LIN {X 0,Y 460.751,Z 770.991,A -85,B 0,C 180,E1 -8393.678,E2 -8393.678} C_VEL
LIN {X 0,Y 461.755,Z 759.273,A -85,B 0,C 180,E1 -8394.503,E2 -8394.503} C_VEL
LIN {X 0,Y 462.708,Z 747.249,A -85,B 0,C 180,E1 -8395.228,E2 -8395.228} C_VEL
LIN {X 0,Y 463.653,Z 734.036,A -85,B 0,C 180,E1 -8395.895,E2 -8395.895} C_VEL
LIN {X 0,Y 464.466,Z 720.83,A -85,B 0,C 180,E1 -8396.438,E2 -8396.438} C_VEL
LIN {X 0,Y 465.142,Z 708.707,A -85,B 0,C 180,E1 -8396.832,E2 -8396.832} C_VEL
LIN {X 0,Y 465.664,Z 695.09,A -85,B 0,C 180,E1 -8397.167,E2 -8397.167} C_VEL
LIN {X 0,Y 466.448,Z 652.564,A -85,B 0,C 180,E1 -8397.875,E2 -8397.875} C_VEL
LIN {X 0,Y 468.618,Z 514.421,A -85,B 0,C 180,E1 -8400.1,E2 -8400.1} C_VEL
LIN {X 0,Y 460.454,Z 482.125,A -85,B 0,C 180,E1 -8401.269,E2 -8401.269} C_VEL
LIN {X 0,Y 460.493,Z 480.391,A -85,B 0,C 180,E1 -8401.488,E2 -8401.488} C_VEL
LIN {X 0,Y 460.182,Z 477.208,A -85,B 0,C 180,E1 -8402.052,E2 -8402.052} C_VEL
LIN {X 0,Y 456.778,Z 463.456,A -85,B 0,C 180,E1 -8404.699,E2 -8404.699} C_VEL
LIN {X 0,Y 453.504,Z 451.445,A -85,B 0,C 180,E1 -8407.184,E2 -8407.184} C_VEL
LIN {X 0,Y 453.456,Z 451.209,A -85,B 0,C 180,E1 -8408.311,E2 -8408.311} C_VEL
LIN {X 0,Y 453.489,Z 451.249,A -85,B 0,C 180,E1 -8410.608,E2 -8410.608} C_VEL
LIN {X 0,Y 453.45,Z 451.247,A -85,B 0,C 180,E1 -8413.243,E2 -8413.243} C_VEL
LIN {X 0,Y 453.471,Z 451.237,A -85,B 0,C 180,E1 -8415.78,E2 -8415.78} C_VEL
LIN {X 0,Y 453.486,Z 451.245,A -85,B 0,C 180,E1 -8418.21,E2 -8418.21} C_VEL
LIN {X 0,Y 453.524,Z 451.233,A -85,B 0,C 180,E1 -8420.787,E2 -8420.787} C_VEL
LIN {X 0,Y 453.45,Z 451.238,A -85,B 0,C 180,E1 -8423.917,E2 -8423.917} C_VEL
LIN {X 0,Y 453.476,Z 451.243,A -85,B 0,C 180,E1 -8427.151,E2 -8427.151} C_VEL
LIN {X 0,Y 453.507,Z 451.223,A -85,B 0,C 180,E1 -8430.271,E2 -8430.271} C_VEL
LIN {X 0,Y 453.506,Z 451.227,A -85,B 0,C 180,E1 -8433.294,E2 -8433.294} C_VEL
LIN {X 0,Y 453.496,Z 451.244,A -85,B 0,C 180,E1 -8436.238,E2 -8436.238} C_VEL
LIN {X 0,Y 453.473,Z 451.215,A -85,B 0,C 180,E1 -8439.117,E2 -8439.117} C_VEL
LIN {X 0,Y 453.502,Z 451.225,A -85,B 0,C 180,E1 -8441.944,E2 -8441.944} C_VEL
LIN {X 0,Y 453.531,Z 451.237,A -85,B 0,C 180,E1 -8444.726,E2 -8444.726} C_VEL
LIN {X 0,Y 453.552,Z 451.239,A -85,B 0,C 180,E1 -8448.379,E2 -8448.379} C_VEL
LIN {X 0,Y 453.643,Z 451.216,A -85,B 0,C 180,E1 -8451.985,E2 -8451.985} C_VEL
LIN {X 0,Y 453.663,Z 451.222,A -85,B 0,C 180,E1 -8454.667,E2 -8454.667} C_VEL
LIN {X 0,Y 453.757,Z 451.205,A -85,B 0,C 180,E1 -8457.337,E2 -8457.337} C_VEL
LIN {X 0,Y 453.814,Z 451.204,A -85,B 0,C 180,E1 -8460,E2 -8460} C_VEL
LIN {X 0,Y 453.757,Z 451.208,A -85,B 0,C 180,E1 -8462.663,E2 -8462.663} C_VEL
LIN {X 0,Y 453.671,Z 451.213,A -85,B 0,C 180,E1 -8466.225,E2 -8466.225} C_VEL
LIN {X 0,Y 453.584,Z 451.232,A -85,B 0,C 180,E1 -8468.913,E2 -8468.913} C_VEL
LIN {X 0,Y 453.554,Z 451.233,A -85,B 0,C 180,E1 -8472.529,E2 -8472.529} C_VEL
LIN {X 0,Y 453.535,Z 451.228,A -85,B 0,C 180,E1 -8476.196,E2 -8476.196} C_VEL
LIN {X 0,Y 453.511,Z 451.24,A -85,B 0,C 180,E1 -8479.041,E2 -8479.041} C_VEL
LIN {X 0,Y 453.467,Z 451.245,A -85,B 0,C 180,E1 -8481.836,E2 -8481.836} C_VEL
LIN {X 0,Y 453.505,Z 451.229,A -85,B 0,C 180,E1 -8484.735,E2 -8484.735} C_VEL
LIN {X 0,Y 453.53,Z 451.223,A -85,B 0,C 180,E1 -8487.961,E2 -8487.961} C_VEL
LIN {X 0,Y 453.475,Z 451.25,A -85,B 0,C 180,E1 -8490.759,E2 -8490.759} C_VEL
LIN {X 0,Y 453.469,Z 451.216,A -85,B 0,C 180,E1 -8493.913,E2 -8493.913} C_VEL
LIN {X 0,Y 453.464,Z 451.253,A -85,B 0,C 180,E1 -8497.188,E2 -8497.188} C_VEL
LIN {X 0,Y 453.525,Z 451.244,A -85,B 0,C 180,E1 -8499.445,E2 -8499.445} C_VEL
LIN {X 0,Y 453.485,Z 451.249,A -85,B 0,C 180,E1 -8502.992,E2 -8502.992} C_VEL
LIN {X 0,Y 453.458,Z 451.251,A -85,B 0,C 180,E1 -8505.779,E2 -8505.779} C_VEL
LIN {X 0,Y 453.509,Z 451.247,A -85,B 0,C 180,E1 -8509.406,E2 -8509.406} C_VEL
LIN {X 0,Y 453.47,Z 451.248,A -85,B 0,C 180,E1 -8512.223,E2 -8512.223} C_VEL
LIN {X 0,Y 453.483,Z 451.25,A -85,B 0,C 180,E1 -8515.223,E2 -8515.223} C_VEL
LIN {X 0,Y 453.461,Z 451.248,A -85,B 0,C 180,E1 -8518.475,E2 -8518.475} C_VEL
LIN {X 0,Y 453.532,Z 451.242,A -85,B 0,C 180,E1 -8522.039,E2 -8522.039} C_VEL
LIN {X 0,Y 453.51,Z 451.246,A -85,B 0,C 180,E1 -8525.266,E2 -8525.266} C_VEL
LIN {X 0,Y 453.476,Z 451.246,A -85,B 0,C 180,E1 -8528.415,E2 -8528.415} C_VEL
LIN {X 0,Y 453.518,Z 451.244,A -85,B 0,C 180,E1 -8531.009,E2 -8531.009} C_VEL
LIN {X 0,Y 453.564,Z 451.238,A -85,B 0,C 180,E1 -8533.88,E2 -8533.88} C_VEL
LIN {X 0,Y 453.598,Z 451.234,A -85,B 0,C 180,E1 -8537.472,E2 -8537.472} C_VEL
LIN {X 0,Y 453.589,Z 451.233,A -85,B 0,C 180,E1 -8541.087,E2 -8541.087} C_VEL
LIN {X 0,Y 453.633,Z 451.228,A -85,B 0,C 180,E1 -8543.099,E2 -8543.099} C_VEL
LIN {X 0,Y 452.948,Z 451.315,A -85,B 0,C 180,E1 -8543.839,E2 -8543.839} C_VEL
LIN {X 0,Y 450.001,Z 451.681,A -85,B 0,C 180,E1 -8545.041,E2 -8545.041} C_VEL
LIN {X 0,Y 447.578,Z 451.985,A -85,B 0,C 180,E1 -8546.01,E2 -8546.01} C_VEL
LIN {X 0,Y 446.642,Z 452.099,A -85,B 0,C 180,E1 -8546.761,E2 -8546.761} C_VEL
LIN {X 0,Y 446.623,Z 452.101,A -85,B 0,C 180,E1 -8547.014,E2 -8547.014} C_VEL
LIN {X 0,Y 446.791,Z 452.084,A -85,B 0,C 180,E1 -8550,E2 -8550} C_VEL
LIN {X 0,Y 446.706,Z 452.093,A -85,B 0,C 180,E1 -8552.705,E2 -8552.705} C_VEL
LIN {X 0,Y 446.643,Z 452.1,A -85,B 0,C 180,E1 -8556.324,E2 -8556.324} C_VEL
LIN {X 0,Y 446.535,Z 452.112,A -85,B 0,C 180,E1 -8559.055,E2 -8559.055} C_VEL
LIN {X 0,Y 446.53,Z 452.113,A -85,B 0,C 180,E1 -8562.729,E2 -8562.729} C_VEL
LIN {X 0,Y 446.486,Z 452.122,A -85,B 0,C 180,E1 -8566.459,E2 -8566.459} C_VEL
LIN {X 0,Y 446.465,Z 452.122,A -85,B 0,C 180,E1 -8569.303,E2 -8569.303} C_VEL
LIN {X 0,Y 446.414,Z 452.131,A -85,B 0,C 180,E1 -8572.199,E2 -8572.199} C_VEL
LIN {X 0,Y 446.453,Z 452.122,A -85,B 0,C 180,E1 -8575.152,E2 -8575.152} C_VEL
LIN {X 0,Y 446.479,Z 452.122,A -85,B 0,C 180,E1 -8578.178,E2 -8578.178} C_VEL
LIN {X 0,Y 446.414,Z 452.127,A -85,B 0,C 180,E1 -8581.775,E2 -8581.775} C_VEL
LIN {X 0,Y 446.425,Z 452.128,A -85,B 0,C 180,E1 -8584.522,E2 -8584.522} C_VEL
LIN {X 0,Y 446.43,Z 452.127,A -85,B 0,C 180,E1 -8588.082,E2 -8588.082} C_VEL
LIN {X 0,Y 446.436,Z 452.126,A -85,B 0,C 180,E1 -8590.92,E2 -8590.92} C_VEL
LIN {X 0,Y 446.394,Z 452.129,A -85,B 0,C 180,E1 -8593.846,E2 -8593.846} C_VEL
LIN {X 0,Y 446.439,Z 452.126,A -85,B 0,C 180,E1 -8596.397,E2 -8596.397} C_VEL
LIN {X 0,Y 446.461,Z 452.12,A -85,B 0,C 180,E1 -8599.805,E2 -8599.805} C_VEL
LIN {X 0,Y 446.427,Z 452.125,A -85,B 0,C 180,E1 -8602.124,E2 -8602.124} C_VEL
LIN {X 0,Y 446.421,Z 452.095,A -85,B 0,C 180,E1 -8605.477,E2 -8605.477} C_VEL
LIN {X 0,Y 446.411,Z 452.125,A -85,B 0,C 180,E1 -8608.7,E2 -8608.7} C_VEL
LIN {X 0,Y 446.476,Z 452.102,A -85,B 0,C 180,E1 -8611.821,E2 -8611.821} C_VEL
LIN {X 0,Y 446.449,Z 452.1,A -85,B 0,C 180,E1 -8614.848,E2 -8614.848} C_VEL
LIN {X 0,Y 446.439,Z 452.121,A -85,B 0,C 180,E1 -8618.245,E2 -8618.245} C_VEL
LIN {X 0,Y 446.448,Z 452.123,A -85,B 0,C 180,E1 -8621.649,E2 -8621.649} C_VEL
LIN {X 0,Y 446.499,Z 452.103,A -85,B 0,C 180,E1 -8624.48,E2 -8624.48} C_VEL
LIN {X 0,Y 446.509,Z 452.104,A -85,B 0,C 180,E1 -8628.193,E2 -8628.193} C_VEL
LIN {X 0,Y 446.591,Z 452.1,A -85,B 0,C 180,E1 -8631.858,E2 -8631.858} C_VEL
LIN {X 0,Y 446.641,Z 452.09,A -85,B 0,C 180,E1 -8634.583,E2 -8634.583} C_VEL
LIN {X 0,Y 446.701,Z 452.089,A -85,B 0,C 180,E1 -8637.295,E2 -8637.295} C_VEL
LIN {X 0,Y 446.784,Z 452.08,A -85,B 0,C 180,E1 -8640,E2 -8640} C_VEL
LIN {X 0,Y 446.701,Z 452.085,A -85,B 0,C 180,E1 -8642.706,E2 -8642.706} C_VEL
LIN {X 0,Y 446.637,Z 452.096,A -85,B 0,C 180,E1 -8646.324,E2 -8646.324} C_VEL
LIN {X 0,Y 446.53,Z 452.099,A -85,B 0,C 180,E1 -8649.056,E2 -8649.056} C_VEL
LIN {X 0,Y 446.513,Z 452.104,A -85,B 0,C 180,E1 -8652.73,E2 -8652.73} C_VEL
LIN {X 0,Y 446.488,Z 452.114,A -85,B 0,C 180,E1 -8656.228,E2 -8656.228} C_VEL
LIN {X 0,Y 446.46,Z 452.087,A -85,B 0,C 180,E1 -8659.304,E2 -8659.304} C_VEL
LIN {X 0,Y 446.41,Z 452.112,A -85,B 0,C 180,E1 -8662.2,E2 -8662.2} C_VEL
LIN {X 0,Y 446.451,Z 452.12,A -85,B 0,C 180,E1 -8665.153,E2 -8665.153} C_VEL
LIN {X 0,Y 446.477,Z 452.086,A -85,B 0,C 180,E1 -8668.179,E2 -8668.179} C_VEL
LIN {X 0,Y 446.412,Z 452.124,A -85,B 0,C 180,E1 -8671.301,E2 -8671.301} C_VEL
LIN {X 0,Y 446.423,Z 452.105,A -85,B 0,C 180,E1 -8674.523,E2 -8674.523} C_VEL
LIN {X 0,Y 446.431,Z 452.126,A -85,B 0,C 180,E1 -8678.083,E2 -8678.083} C_VEL
LIN {X 0,Y 446.44,Z 452.116,A -85,B 0,C 180,E1 -8680.921,E2 -8680.921} C_VEL
LIN {X 0,Y 446.44,Z 452.114,A -85,B 0,C 180,E1 -8683.841,E2 -8683.841} C_VEL
LIN {X 0,Y 446.394,Z 452.129,A -85,B 0,C 180,E1 -8686.404,E2 -8686.404} C_VEL
LIN {X 0,Y 446.422,Z 452.13,A -85,B 0,C 180,E1 -8689.083,E2 -8689.083} C_VEL
LIN {X 0,Y 446.432,Z 452.17,A -85,B 0,C 180,E1 -8692.267,E2 -8692.267} C_VEL
LIN {X 0,Y 446.953,Z 454.055,A -85,B 0,C 180,E1 -8692.745,E2 -8692.745} C_VEL
LIN {X 0,Y 451.035,Z 469.273,A -85,B 0,C 180,E1 -8695.879,E2 -8695.879} C_VEL
LIN {X 0,Y 453.742,Z 480.765,A -85,B 0,C 180,E1 -8698.093,E2 -8698.093} C_VEL
LIN {X 0,Y 453.963,Z 482.255,A -85,B 0,C 180,E1 -8698.24,E2 -8698.24} C_VEL
LIN {X 0,Y 460.479,Z 508.061,A -85,B 0,C 180,E1 -8699.203,E2 -8699.203} C_VEL
LIN {X 0,Y 462.541,Z 516.964,A -85,B 0,C 180,E1 -8699.511,E2 -8699.511} C_VEL
LIN {X 0,Y 459.412,Z 692.172,A -85,B 0,C 180,E1 -8702.374,E2 -8702.374} C_VEL
LIN {X 0,Y 458.878,Z 705.317,A -85,B 0,C 180,E1 -8702.674,E2 -8702.674} C_VEL
LIN {X 0,Y 458.235,Z 718.558,A -85,B 0,C 180,E1 -8703.091,E2 -8703.091} C_VEL
LIN {X 0,Y 457.427,Z 731.356,A -85,B 0,C 180,E1 -8703.603,E2 -8703.603} C_VEL
LIN {X 0,Y 456.547,Z 743.961,A -85,B 0,C 180,E1 -8704.223,E2 -8704.223} C_VEL
LIN {X 0,Y 455.579,Z 755.577,A -85,B 0,C 180,E1 -8704.899,E2 -8704.899} C_VEL
LIN {X 0,Y 454.543,Z 767.509,A -85,B 0,C 180,E1 -8705.714,E2 -8705.714} C_VEL
LIN {X 0,Y 453.327,Z 780.062,A -85,B 0,C 180,E1 -8706.714,E2 -8706.714} C_VEL
LIN {X 0,Y 452.325,Z 790.059,A -85,B 0,C 180,E1 -8707.625,E2 -8707.625} C_VEL
LIN {X 0,Y 451.186,Z 801.044,A -85,B 0,C 180,E1 -8708.768,E2 -8708.768} C_VEL
LIN {X 0,Y 450.195,Z 810.74,A -85,B 0,C 180,E1 -8709.914,E2 -8709.914} C_VEL
LIN {X 0,Y 449.109,Z 820.953,A -85,B 0,C 180,E1 -8711.289,E2 -8711.289} C_VEL
LIN {X 0,Y 448.266,Z 829.916,A -85,B 0,C 180,E1 -8712.67,E2 -8712.67} C_VEL
LIN {X 0,Y 447.597,Z 837.811,A -85,B 0,C 180,E1 -8714.052,E2 -8714.052} C_VEL
LIN {X 0,Y 446.972,Z 844.773,A -85,B 0,C 180,E1 -8715.429,E2 -8715.429} C_VEL
LIN {X 0,Y 446.534,Z 850.913,A -85,B 0,C 180,E1 -8716.808,E2 -8716.808} C_VEL
LIN {X 0,Y 446.02,Z 857.853,A -85,B 0,C 180,E1 -8718.641,E2 -8718.641} C_VEL
LIN {X 0,Y 445.675,Z 863.601,A -85,B 0,C 180,E1 -8720.469,E2 -8720.469} C_VEL
LIN {X 0,Y 445.568,Z 867.207,A -85,B 0,C 180,E1 -8721.839,E2 -8721.839} C_VEL
LIN {X 0,Y 445.487,Z 871.048,A -85,B 0,C 180,E1 -8723.66,E2 -8723.66} C_VEL
LIN {X 0,Y 445.362,Z 873.884,A -85,B 0,C 180,E1 -8725.475,E2 -8725.475} C_VEL
LIN {X 0,Y 445.406,Z 875.76,A -85,B 0,C 180,E1 -8727.287,E2 -8727.287} C_VEL
LIN {X 0,Y 445.346,Z 876.431,A -85,B 0,C 180,E1 -8728.191,E2 -8728.191} C_VEL
LIN {X 0,Y 445.287,Z 876.899,A -85,B 0,C 180,E1 -8730,E2 -8730} C_VEL
LIN {X 0,Y 445.346,Z 876.431,A -85,B 0,C 180,E1 -8731.809,E2 -8731.809} C_VEL
LIN {X 0,Y 445.331,Z 875.014,A -85,B 0,C 180,E1 -8733.619,E2 -8733.619} C_VEL
LIN {X 0,Y 445.402,Z 872.641,A -85,B 0,C 180,E1 -8735.432,E2 -8735.432} C_VEL
LIN {X 0,Y 445.537,Z 868.244,A -85,B 0,C 180,E1 -8737.705,E2 -8737.705} C_VEL
LIN {X 0,Y 445.637,Z 864.885,A -85,B 0,C 180,E1 -8739.074,E2 -8739.074} C_VEL
LIN {X 0,Y 445.932,Z 859.395,A -85,B 0,C 180,E1 -8740.901,E2 -8740.901} C_VEL
LIN {X 0,Y 446.257,Z 853.787,A -85,B 0,C 180,E1 -8742.467,E2 -8742.467} C_VEL
LIN {X 0,Y 446.774,Z 846.878,A -85,B 0,C 180,E1 -8744.112,E2 -8744.112} C_VEL
LIN {X 0,Y 447.367,Z 840.229,A -85,B 0,C 180,E1 -8745.489,E2 -8745.489} C_VEL
LIN {X 0,Y 448.044,Z 832.524,A -85,B 0,C 180,E1 -8746.895,E2 -8746.895} C_VEL
LIN {X 0,Y 448.789,Z 824.086,A -85,B 0,C 180,E1 -8748.252,E2 -8748.252} C_VEL
LIN {X 0,Y 449.804,Z 814.293,A -85,B 0,C 180,E1 -8749.629,E2 -8749.629} C_VEL
LIN {X 0,Y 450.829,Z 804.634,A -85,B 0,C 180,E1 -8750.824,E2 -8750.824} C_VEL
LIN {X 0,Y 451.954,Z 793.492,A -85,B 0,C 180,E1 -8752.033,E2 -8752.033} C_VEL
LIN {X 0,Y 453.028,Z 782.673,A -85,B 0,C 180,E1 -8753.061,E2 -8753.061} C_VEL
LIN {X 0,Y 454.193,Z 770.779,A -85,B 0,C 180,E1 -8754.041,E2 -8754.041} C_VEL
LIN {X 0,Y 455.242,Z 759.061,A -85,B 0,C 180,E1 -8754.877,E2 -8754.877} C_VEL
LIN {X 0,Y 456.249,Z 747.038,A -85,B 0,C 180,E1 -8755.611,E2 -8755.611} C_VEL
LIN {X 0,Y 457.254,Z 733.826,A -85,B 0,C 180,E1 -8756.285,E2 -8756.285} C_VEL
LIN {X 0,Y 458.113,Z 720.656,A -85,B 0,C 180,E1 -8756.832,E2 -8756.832} C_VEL
LIN {X 0,Y 458.805,Z 708.409,A -85,B 0,C 180,E1 -8757.235,E2 -8757.235} C_VEL
LIN {X 0,Y 459.336,Z 695.012,A -85,B 0,C 180,E1 -8757.57,E2 -8757.57} C_VEL
LIN {X 0,Y 460.05,Z 659.518,A -85,B 0,C 180,E1 -8758.173,E2 -8758.173} C_VEL
LIN {X 0,Y 462.503,Z 516.907,A -85,B 0,C 180,E1 -8760.493,E2 -8760.493} C_VEL
LIN {X 0,Y 457.598,Z 496.123,A -85,B 0,C 180,E1 -8761.224,E2 -8761.224} C_VEL
LIN {X 0,Y 453.81,Z 481.493,A -85,B 0,C 180,E1 -8761.804,E2 -8761.804} C_VEL
LIN {X 0,Y 452.155,Z 473.861,A -85,B 0,C 180,E1 -8763.222,E2 -8763.222} C_VEL
LIN {X 0,Y 448.771,Z 460.638,A -85,B 0,C 180,E1 -8765.862,E2 -8765.862} C_VEL
LIN {X 0,Y 446.49,Z 452.566,A -85,B 0,C 180,E1 -8767.584,E2 -8767.584} C_VEL
LIN {X 0,Y 446.403,Z 452.091,A -85,B 0,C 180,E1 -8767.878,E2 -8767.878} C_VEL
LIN {X 0,Y 446.422,Z 452.13,A -85,B 0,C 180,E1 -8770.917,E2 -8770.917} C_VEL
LIN {X 0,Y 446.412,Z 452.132,A -85,B 0,C 180,E1 -8773.843,E2 -8773.843} C_VEL
LIN {X 0,Y 446.441,Z 452.116,A -85,B 0,C 180,E1 -8776.396,E2 -8776.396} C_VEL
LIN {X 0,Y 446.462,Z 452.107,A -85,B 0,C 180,E1 -8779.804,E2 -8779.804} C_VEL
LIN {X 0,Y 446.427,Z 452.128,A -85,B 0,C 180,E1 -8782.123,E2 -8782.123} C_VEL
LIN {X 0,Y 446.423,Z 452.105,A -85,B 0,C 180,E1 -8785.477,E2 -8785.477} C_VEL
LIN {X 0,Y 446.412,Z 452.124,A -85,B 0,C 180,E1 -8788.699,E2 -8788.699} C_VEL
LIN {X 0,Y 446.477,Z 452.086,A -85,B 0,C 180,E1 -8791.821,E2 -8791.821} C_VEL
LIN {X 0,Y 446.451,Z 452.12,A -85,B 0,C 180,E1 -8794.847,E2 -8794.847} C_VEL
LIN {X 0,Y 446.44,Z 452.099,A -85,B 0,C 180,E1 -8798.245,E2 -8798.245} C_VEL
LIN {X 0,Y 446.448,Z 452.099,A -85,B 0,C 180,E1 -8801.649,E2 -8801.649} C_VEL
LIN {X 0,Y 446.499,Z 452.116,A -85,B 0,C 180,E1 -8804.479,E2 -8804.479} C_VEL
LIN {X 0,Y 446.51,Z 452.112,A -85,B 0,C 180,E1 -8808.193,E2 -8808.193} C_VEL
LIN {X 0,Y 446.591,Z 452.093,A -85,B 0,C 180,E1 -8811.858,E2 -8811.858} C_VEL
LIN {X 0,Y 446.637,Z 452.098,A -85,B 0,C 180,E1 -8814.582,E2 -8814.582} C_VEL
LIN {X 0,Y 446.701,Z 452.084,A -85,B 0,C 180,E1 -8817.294,E2 -8817.294} C_VEL
LIN {X 0,Y 446.784,Z 452.079,A -85,B 0,C 180,E1 -8820,E2 -8820} C_VEL
LIN {X 0,Y 446.701,Z 452.088,A -85,B 0,C 180,E1 -8822.705,E2 -8822.705} C_VEL
LIN {X 0,Y 446.64,Z 452.088,A -85,B 0,C 180,E1 -8826.324,E2 -8826.324} C_VEL
LIN {X 0,Y 446.53,Z 452.109,A -85,B 0,C 180,E1 -8829.055,E2 -8829.055} C_VEL
LIN {X 0,Y 446.512,Z 452.113,A -85,B 0,C 180,E1 -8832.73,E2 -8832.73} C_VEL
LIN {X 0,Y 446.487,Z 452.106,A -85,B 0,C 180,E1 -8836.228,E2 -8836.228} C_VEL
LIN {X 0,Y 446.46,Z 452.116,A -85,B 0,C 180,E1 -8839.303,E2 -8839.303} C_VEL
LIN {X 0,Y 446.409,Z 452.126,A -85,B 0,C 180,E1 -8842.2,E2 -8842.2} C_VEL
LIN {X 0,Y 446.449,Z 452.1,A -85,B 0,C 180,E1 -8845.152,E2 -8845.152} C_VEL
LIN {X 0,Y 446.476,Z 452.102,A -85,B 0,C 180,E1 -8848.179,E2 -8848.179} C_VEL
LIN {X 0,Y 446.411,Z 452.125,A -85,B 0,C 180,E1 -8851.3,E2 -8851.3} C_VEL
LIN {X 0,Y 446.421,Z 452.095,A -85,B 0,C 180,E1 -8854.523,E2 -8854.523} C_VEL
LIN {X 0,Y 446.431,Z 452.124,A -85,B 0,C 180,E1 -8858.083,E2 -8858.083} C_VEL
LIN {X 0,Y 446.44,Z 452.127,A -85,B 0,C 180,E1 -8860.921,E2 -8860.921} C_VEL
LIN {X 0,Y 446.438,Z 452.124,A -85,B 0,C 180,E1 -8863.841,E2 -8863.841} C_VEL
LIN {X 0,Y 446.392,Z 452.129,A -85,B 0,C 180,E1 -8866.404,E2 -8866.404} C_VEL
LIN {X 0,Y 446.461,Z 452.122,A -85,B 0,C 180,E1 -8869.805,E2 -8869.805} C_VEL
LIN {X 0,Y 446.426,Z 452.126,A -85,B 0,C 180,E1 -8872.124,E2 -8872.124} C_VEL
LIN {X 0,Y 446.425,Z 452.128,A -85,B 0,C 180,E1 -8875.478,E2 -8875.478} C_VEL
LIN {X 0,Y 446.411,Z 452.127,A -85,B 0,C 180,E1 -8878.7,E2 -8878.7} C_VEL
LIN {X 0,Y 446.479,Z 452.121,A -85,B 0,C 180,E1 -8881.822,E2 -8881.822} C_VEL
LIN {X 0,Y 446.453,Z 452.122,A -85,B 0,C 180,E1 -8884.848,E2 -8884.848} C_VEL
LIN {X 0,Y 446.444,Z 452.123,A -85,B 0,C 180,E1 -8888.245,E2 -8888.245} C_VEL
LIN {X 0,Y 446.453,Z 452.124,A -85,B 0,C 180,E1 -8891.649,E2 -8891.649} C_VEL
LIN {X 0,Y 446.504,Z 452.118,A -85,B 0,C 180,E1 -8894.48,E2 -8894.48} C_VEL
LIN {X 0,Y 446.536,Z 452.113,A -85,B 0,C 180,E1 -8898.194,E2 -8898.194} C_VEL
LIN {X 0,Y 446.597,Z 452.108,A -85,B 0,C 180,E1 -8901.858,E2 -8901.858} C_VEL
LIN {X 0,Y 446.642,Z 452.1,A -85,B 0,C 180,E1 -8904.583,E2 -8904.583} C_VEL
LIN {X 0,Y 446.623,Z 452.101,A -85,B 0,C 180,E1 -8907.014,E2 -8907.014} C_VEL
LIN {X 0,Y 446.105,Z 452.169,A -85,B 0,C 180,E1 -8907.767,E2 -8907.767} C_VEL
LIN {X 0,Y 443.287,Z 452.522,A -85,B 0,C 180,E1 -8908.99,E2 -8908.99} C_VEL
LIN {X 0,Y 440.8,Z 452.831,A -85,B 0,C 180,E1 -8909.977,E2 -8909.977} C_VEL
LIN {X 0,Y 439.712,Z 452.964,A -85,B 0,C 180,E1 -8910.74,E2 -8910.74} C_VEL
LIN {X 0,Y 439.618,Z 452.974,A -85,B 0,C 180,E1 -8910.999,E2 -8910.999} C_VEL
LIN {X 0,Y 439.653,Z 452.971,A -85,B 0,C 180,E1 -8912.749,E2 -8912.749} C_VEL
LIN {X 0,Y 439.614,Z 452.976,A -85,B 0,C 180,E1 -8916.425,E2 -8916.425} C_VEL
LIN {X 0,Y 439.497,Z 452.989,A -85,B 0,C 180,E1 -8919.201,E2 -8919.201} C_VEL
LIN {X 0,Y 439.5,Z 452.989,A -85,B 0,C 180,E1 -8922.726,E2 -8922.726} C_VEL
LIN {X 0,Y 439.443,Z 452.998,A -85,B 0,C 180,E1 -8926.349,E2 -8926.349} C_VEL
LIN {X 0,Y 439.398,Z 453.003,A -85,B 0,C 180,E1 -8929.626,E2 -8929.626} C_VEL
LIN {X 0,Y 439.36,Z 453.007,A -85,B 0,C 180,E1 -8932.575,E2 -8932.575} C_VEL
LIN {X 0,Y 439.4,Z 453,A -85,B 0,C 180,E1 -8935.585,E2 -8935.585} C_VEL
LIN {X 0,Y 439.412,Z 453.001,A -85,B 0,C 180,E1 -8938.673,E2 -8938.673} C_VEL
LIN {X 0,Y 439.365,Z 453.007,A -85,B 0,C 180,E1 -8942.03,E2 -8942.03} C_VEL
LIN {X 0,Y 439.39,Z 453,A -85,B 0,C 180,E1 -8945.34,E2 -8945.34} C_VEL
LIN {X 0,Y 439.391,Z 453.004,A -85,B 0,C 180,E1 -8948.593,E2 -8948.593} C_VEL
LIN {X 0,Y 439.391,Z 453.002,A -85,B 0,C 180,E1 -8951.258,E2 -8951.258} C_VEL
LIN {X 0,Y 439.395,Z 453.004,A -85,B 0,C 180,E1 -8954.729,E2 -8954.729} C_VEL
LIN {X 0,Y 439.405,Z 452.999,A -85,B 0,C 180,E1 -8957.797,E2 -8957.797} C_VEL
LIN {X 0,Y 439.444,Z 452.996,A -85,B 0,C 180,E1 -8960.23,E2 -8960.23} C_VEL
LIN {X 0,Y 439.369,Z 452.999,A -85,B 0,C 180,E1 -8963.713,E2 -8963.713} C_VEL
LIN {X 0,Y 439.364,Z 452.981,A -85,B 0,C 180,E1 -8967.054,E2 -8967.054} C_VEL
LIN {X 0,Y 439.388,Z 453.001,A -85,B 0,C 180,E1 -8970.275,E2 -8970.275} C_VEL
LIN {X 0,Y 439.425,Z 452.962,A -85,B 0,C 180,E1 -8973.588,E2 -8973.588} C_VEL
LIN {X 0,Y 439.377,Z 452.998,A -85,B 0,C 180,E1 -8976.429,E2 -8976.429} C_VEL
LIN {X 0,Y 439.379,Z 452.996,A -85,B 0,C 180,E1 -8979.397,E2 -8979.397} C_VEL
LIN {X 0,Y 439.422,Z 452.995,A -85,B 0,C 180,E1 -8982.309,E2 -8982.309} C_VEL
LIN {X 0,Y 439.439,Z 452.989,A -85,B 0,C 180,E1 -8985.174,E2 -8985.174} C_VEL
LIN {X 0,Y 439.475,Z 452.981,A -85,B 0,C 180,E1 -8988.001,E2 -8988.001} C_VEL
LIN {X 0,Y 439.539,Z 452.98,A -85,B 0,C 180,E1 -8991.726,E2 -8991.726} C_VEL
LIN {X 0,Y 439.616,Z 452.965,A -85,B 0,C 180,E1 -8994.496,E2 -8994.496} C_VEL
LIN {X 0,Y 439.627,Z 452.959,A -85,B 0,C 180,E1 -8998.168,E2 -8998.168} C_VEL
LIN {X 0,Y 439.754,Z 452.956,A -85,B 0,C 180,E1 -9000,E2 -9000} C_VEL
LIN {X 0,Y 439.648,Z 452.964,A -85,B 0,C 180,E1 -9002.749,E2 -9002.749} C_VEL
LIN {X 0,Y 439.609,Z 452.971,A -85,B 0,C 180,E1 -9006.425,E2 -9006.425} C_VEL
LIN {X 0,Y 439.492,Z 452.977,A -85,B 0,C 180,E1 -9009.202,E2 -9009.202} C_VEL
LIN {X 0,Y 439.457,Z 452.984,A -85,B 0,C 180,E1 -9012.938,E2 -9012.938} C_VEL
LIN {X 0,Y 439.439,Z 452.991,A -85,B 0,C 180,E1 -9016.349,E2 -9016.349} C_VEL
LIN {X 0,Y 439.394,Z 452.962,A -85,B 0,C 180,E1 -9019.627,E2 -9019.627} C_VEL
LIN {X 0,Y 439.357,Z 452.998,A -85,B 0,C 180,E1 -9022.576,E2 -9022.576} C_VEL
LIN {X 0,Y 439.398,Z 452.999,A -85,B 0,C 180,E1 -9025.585,E2 -9025.585} C_VEL
LIN {X 0,Y 439.418,Z 452.965,A -85,B 0,C 180,E1 -9028.673,E2 -9028.673} C_VEL
LIN {X 0,Y 439.376,Z 453.008,A -85,B 0,C 180,E1 -9032.034,E2 -9032.034} C_VEL
LIN {X 0,Y 439.389,Z 452.98,A -85,B 0,C 180,E1 -9035.341,E2 -9035.341} C_VEL
LIN {X 0,Y 439.391,Z 452.996,A -85,B 0,C 180,E1 -9038.594,E2 -9038.594} C_VEL
LIN {X 0,Y 439.397,Z 452.997,A -85,B 0,C 180,E1 -9041.26,E2 -9041.26} C_VEL
LIN {X 0,Y 439.403,Z 452.99,A -85,B 0,C 180,E1 -9044.729,E2 -9044.729} C_VEL
LIN {X 0,Y 439.391,Z 452.991,A -85,B 0,C 180,E1 -9047.796,E2 -9047.796} C_VEL
LIN {X 0,Y 439.384,Z 452.984,A -85,B 0,C 180,E1 -9050.224,E2 -9050.224} C_VEL
LIN {X 0,Y 439.371,Z 453.063,A -85,B 0,C 180,E1 -9051.771,E2 -9051.771} C_VEL
LIN {X 0,Y 439.513,Z 453.763,A -85,B 0,C 180,E1 -9052.004,E2 -9052.004} C_VEL
LIN {X 0,Y 443.327,Z 467.493,A -85,B 0,C 180,E1 -9054.935,E2 -9054.935} C_VEL
LIN {X 0,Y 446.762,Z 481.269,A -85,B 0,C 180,E1 -9057.638,E2 -9057.638} C_VEL
LIN {X 0,Y 448.587,Z 486.422,A -85,B 0,C 180,E1 -9057.902,E2 -9057.902} C_VEL
LIN {X 0,Y 456.38,Z 517.644,A -85,B 0,C 180,E1 -9059.07,E2 -9059.07} C_VEL
LIN {X 0,Y 453.241,Z 689.123,A -85,B 0,C 180,E1 -9061.902,E2 -9061.902} C_VEL
LIN {X 0,Y 452.592,Z 704.257,A -85,B 0,C 180,E1 -9062.235,E2 -9062.235} C_VEL
LIN {X 0,Y 451.908,Z 717.826,A -85,B 0,C 180,E1 -9062.662,E2 -9062.662} C_VEL
LIN {X 0,Y 451.041,Z 731.145,A -85,B 0,C 180,E1 -9063.199,E2 -9063.199} C_VEL
LIN {X 0,Y 450.193,Z 742.722,A -85,B 0,C 180,E1 -9063.77,E2 -9063.77} C_VEL
LIN {X 0,Y 449.093,Z 755.365,A -85,B 0,C 180,E1 -9064.51,E2 -9064.51} C_VEL
LIN {X 0,Y 447.916,Z 768.267,A -85,B 0,C 180,E1 -9065.411,E2 -9065.411} C_VEL
LIN {X 0,Y 446.748,Z 779.85,A -85,B 0,C 180,E1 -9066.35,E2 -9066.35} C_VEL
LIN {X 0,Y 445.647,Z 789.845,A -85,B 0,C 180,E1 -9067.272,E2 -9067.272} C_VEL
LIN {X 0,Y 444.432,Z 800.829,A -85,B 0,C 180,E1 -9068.429,E2 -9068.429} C_VEL
LIN {X 0,Y 443.419,Z 810.527,A -85,B 0,C 180,E1 -9069.593,E2 -9069.593} C_VEL
LIN {X 0,Y 442.273,Z 820.739,A -85,B 0,C 180,E1 -9070.989,E2 -9070.989} C_VEL
LIN {X 0,Y 441.345,Z 829.701,A -85,B 0,C 180,E1 -9072.389,E2 -9072.389} C_VEL
LIN {X 0,Y 440.668,Z 837.598,A -85,B 0,C 180,E1 -9073.794,E2 -9073.794} C_VEL
LIN {X 0,Y 439.971,Z 844.56,A -85,B 0,C 180,E1 -9075.192,E2 -9075.192} C_VEL
LIN {X 0,Y 439.522,Z 850.701,A -85,B 0,C 180,E1 -9076.594,E2 -9076.594} C_VEL
LIN {X 0,Y 438.975,Z 857.641,A -85,B 0,C 180,E1 -9078.456,E2 -9078.456} C_VEL
LIN {X 0,Y 438.605,Z 863.389,A -85,B 0,C 180,E1 -9080.314,E2 -9080.314} C_VEL
LIN {X 0,Y 438.477,Z 866.996,A -85,B 0,C 180,E1 -9081.706,E2 -9081.706} C_VEL
LIN {X 0,Y 438.393,Z 871.062,A -85,B 0,C 180,E1 -9083.687,E2 -9083.687} C_VEL
LIN {X 0,Y 438.284,Z 873.675,A -85,B 0,C 180,E1 -9085.401,E2 -9085.401} C_VEL
LIN {X 0,Y 438.313,Z 875.55,A -85,B 0,C 180,E1 -9087.243,E2 -9087.243} C_VEL
LIN {X 0,Y 438.268,Z 876.221,A -85,B 0,C 180,E1 -9088.162,E2 -9088.162} C_VEL
LIN {X 0,Y 438.201,Z 876.689,A -85,B 0,C 180,E1 -9090,E2 -9090} C_VEL
LIN {X 0,Y 438.268,Z 876.221,A -85,B 0,C 180,E1 -9091.838,E2 -9091.838} C_VEL
LIN {X 0,Y 438.234,Z 874.804,A -85,B 0,C 180,E1 -9093.678,E2 -9093.678} C_VEL
LIN {X 0,Y 438.31,Z 872.431,A -85,B 0,C 180,E1 -9095.521,E2 -9095.521} C_VEL
LIN {X 0,Y 438.476,Z 869.071,A -85,B 0,C 180,E1 -9097.367,E2 -9097.367} C_VEL
LIN {X 0,Y 438.568,Z 864.673,A -85,B 0,C 180,E1 -9099.221,E2 -9099.221} C_VEL
LIN {X 0,Y 438.89,Z 859.183,A -85,B 0,C 180,E1 -9101.078,E2 -9101.078} C_VEL
LIN {X 0,Y 439.219,Z 853.997,A -85,B 0,C 180,E1 -9102.561,E2 -9102.561} C_VEL
LIN {X 0,Y 439.793,Z 846.665,A -85,B 0,C 180,E1 -9104.341,E2 -9104.341} C_VEL
LIN {X 0,Y 440.433,Z 840.016,A -85,B 0,C 180,E1 -9105.739,E2 -9105.739} C_VEL
LIN {X 0,Y 441.148,Z 832.039,A -85,B 0,C 180,E1 -9107.214,E2 -9107.214} C_VEL
LIN {X 0,Y 441.933,Z 823.873,A -85,B 0,C 180,E1 -9108.545,E2 -9108.545} C_VEL
LIN {X 0,Y 443.014,Z 814.08,A -85,B 0,C 180,E1 -9109.942,E2 -9109.942} C_VEL
LIN {X 0,Y 444.109,Z 803.843,A -85,B 0,C 180,E1 -9111.223,E2 -9111.223} C_VEL
LIN {X 0,Y 445.285,Z 793.279,A -85,B 0,C 180,E1 -9112.381,E2 -9112.381} C_VEL
LIN {X 0,Y 446.43,Z 782.46,A -85,B 0,C 180,E1 -9113.422,E2 -9113.422} C_VEL
LIN {X 0,Y 447.636,Z 770.642,A -85,B 0,C 180,E1 -9114.41,E2 -9114.41} C_VEL
LIN {X 0,Y 448.762,Z 758.85,A -85,B 0,C 180,E1 -9115.261,E2 -9115.261} C_VEL
LIN {X 0,Y 449.807,Z 746.827,A -85,B 0,C 180,E1 -9116.005,E2 -9116.005} C_VEL
LIN {X 0,Y 450.874,Z 733.615,A -85,B 0,C 180,E1 -9116.686,E2 -9116.686} C_VEL
LIN {X 0,Y 451.72,Z 721.008,A -85,B 0,C 180,E1 -9117.22,E2 -9117.22} C_VEL
LIN {X 0,Y 452.485,Z 708.368,A -85,B 0,C 180,E1 -9117.643,E2 -9117.643} C_VEL
LIN {X 0,Y 453.056,Z 694.802,A -85,B 0,C 180,E1 -9117.985,E2 -9117.985} C_VEL
LIN {X 0,Y 453.816,Z 657.517,A -85,B 0,C 180,E1 -9118.627,E2 -9118.627} C_VEL
LIN {X 0,Y 456.348,Z 518.344,A -85,B 0,C 180,E1 -9120.92,E2 -9120.92} C_VEL
LIN {X 0,Y 453.179,Z 504.27,A -85,B 0,C 180,E1 -9121.413,E2 -9121.413} C_VEL
LIN {X 0,Y 447.914,Z 484.156,A -85,B 0,C 180,E1 -9122.193,E2 -9122.193} C_VEL
LIN {X 0,Y 446.683,Z 481.143,A -85,B 0,C 180,E1 -9122.379,E2 -9122.379} C_VEL
LIN {X 0,Y 443.707,Z 468.969,A -85,B 0,C 180,E1 -9124.764,E2 -9124.764} C_VEL
LIN {X 0,Y 440.423,Z 456.801,A -85,B 0,C 180,E1 -9127.327,E2 -9127.327} C_VEL
LIN {X 0,Y 439.411,Z 453.205,A -85,B 0,C 180,E1 -9128.152,E2 -9128.152} C_VEL
LIN {X 0,Y 439.366,Z 452.962,A -85,B 0,C 180,E1 -9128.596,E2 -9128.596} C_VEL
LIN {X 0,Y 439.383,Z 453.002,A -85,B 0,C 180,E1 -9131.256,E2 -9131.256} C_VEL
LIN {X 0,Y 439.399,Z 452.998,A -85,B 0,C 180,E1 -9134.728,E2 -9134.728} C_VEL
LIN {X 0,Y 439.404,Z 453.004,A -85,B 0,C 180,E1 -9137.797,E2 -9137.797} C_VEL
LIN {X 0,Y 439.445,Z 452.98,A -85,B 0,C 180,E1 -9140.229,E2 -9140.229} C_VEL
LIN {X 0,Y 439.371,Z 452.994,A -85,B 0,C 180,E1 -9143.713,E2 -9143.713} C_VEL
LIN {X 0,Y 439.368,Z 453,A -85,B 0,C 180,E1 -9147.054,E2 -9147.054} C_VEL
LIN {X 0,Y 439.388,Z 452.98,A -85,B 0,C 180,E1 -9150.275,E2 -9150.275} C_VEL
LIN {X 0,Y 439.423,Z 452.981,A -85,B 0,C 180,E1 -9153.396,E2 -9153.396} C_VEL
LIN {X 0,Y 439.379,Z 453,A -85,B 0,C 180,E1 -9156.429,E2 -9156.429} C_VEL
LIN {X 0,Y 439.379,Z 452.964,A -85,B 0,C 180,E1 -9159.397,E2 -9159.397} C_VEL
LIN {X 0,Y 439.423,Z 452.983,A -85,B 0,C 180,E1 -9162.309,E2 -9162.309} C_VEL
LIN {X 0,Y 439.439,Z 452.991,A -85,B 0,C 180,E1 -9165.174,E2 -9165.174} C_VEL
LIN {X 0,Y 439.476,Z 452.986,A -85,B 0,C 180,E1 -9168.001,E2 -9168.001} C_VEL
LIN {X 0,Y 439.539,Z 452.97,A -85,B 0,C 180,E1 -9171.726,E2 -9171.726} C_VEL
LIN {X 0,Y 439.613,Z 452.974,A -85,B 0,C 180,E1 -9174.496,E2 -9174.496} C_VEL
LIN {X 0,Y 439.627,Z 452.97,A -85,B 0,C 180,E1 -9178.168,E2 -9178.168} C_VEL
LIN {X 0,Y 439.754,Z 452.955,A -85,B 0,C 180,E1 -9180,E2 -9180} C_VEL
LIN {X 0,Y 439.648,Z 452.966,A -85,B 0,C 180,E1 -9182.749,E2 -9182.749} C_VEL
LIN {X 0,Y 439.611,Z 452.963,A -85,B 0,C 180,E1 -9186.425,E2 -9186.425} C_VEL
LIN {X 0,Y 439.492,Z 452.984,A -85,B 0,C 180,E1 -9189.202,E2 -9189.202} C_VEL
LIN {X 0,Y 439.456,Z 452.995,A -85,B 0,C 180,E1 -9192.938,E2 -9192.938} C_VEL
LIN {X 0,Y 439.438,Z 452.985,A -85,B 0,C 180,E1 -9196.349,E2 -9196.349} C_VEL
LIN {X 0,Y 439.393,Z 452.994,A -85,B 0,C 180,E1 -9199.626,E2 -9199.626} C_VEL
LIN {X 0,Y 439.356,Z 453.008,A -85,B 0,C 180,E1 -9202.576,E2 -9202.576} C_VEL
LIN {X 0,Y 439.396,Z 452.974,A -85,B 0,C 180,E1 -9205.585,E2 -9205.585} C_VEL
LIN {X 0,Y 439.417,Z 452.984,A -85,B 0,C 180,E1 -9208.673,E2 -9208.673} C_VEL
LIN {X 0,Y 439.366,Z 452.998,A -85,B 0,C 180,E1 -9211.861,E2 -9211.861} C_VEL
LIN {X 0,Y 439.392,Z 452.977,A -85,B 0,C 180,E1 -9215.156,E2 -9215.156} C_VEL
LIN {X 0,Y 439.391,Z 453.003,A -85,B 0,C 180,E1 -9218.594,E2 -9218.594} C_VEL
LIN {X 0,Y 439.398,Z 453.005,A -85,B 0,C 180,E1 -9221.26,E2 -9221.26} C_VEL
LIN {X 0,Y 439.401,Z 453.002,A -85,B 0,C 180,E1 -9224.729,E2 -9224.729} C_VEL
LIN {X 0,Y 439.39,Z 453.003,A -85,B 0,C 180,E1 -9227.796,E2 -9227.796} C_VEL
LIN {X 0,Y 439.444,Z 452.995,A -85,B 0,C 180,E1 -9230.23,E2 -9230.23} C_VEL
LIN {X 0,Y 439.371,Z 453.006,A -85,B 0,C 180,E1 -9233.714,E2 -9233.714} C_VEL
LIN {X 0,Y 439.367,Z 453.007,A -85,B 0,C 180,E1 -9237.054,E2 -9237.054} C_VEL
LIN {X 0,Y 439.377,Z 453.004,A -85,B 0,C 180,E1 -9240.275,E2 -9240.275} C_VEL
LIN {X 0,Y 439.425,Z 452.999,A -85,B 0,C 180,E1 -9243.397,E2 -9243.397} C_VEL
LIN {X 0,Y 439.382,Z 453.004,A -85,B 0,C 180,E1 -9246.43,E2 -9246.43} C_VEL
LIN {X 0,Y 439.384,Z 453.007,A -85,B 0,C 180,E1 -9249.397,E2 -9249.397} C_VEL
LIN {X 0,Y 439.427,Z 452.998,A -85,B 0,C 180,E1 -9252.31,E2 -9252.31} C_VEL
LIN {X 0,Y 439.444,Z 452.998,A -85,B 0,C 180,E1 -9255.174,E2 -9255.174} C_VEL
LIN {X 0,Y 439.504,Z 452.989,A -85,B 0,C 180,E1 -9258.002,E2 -9258.002} C_VEL
LIN {X 0,Y 439.545,Z 452.986,A -85,B 0,C 180,E1 -9261.726,E2 -9261.726} C_VEL
LIN {X 0,Y 439.617,Z 452.976,A -85,B 0,C 180,E1 -9264.496,E2 -9264.496} C_VEL
LIN {X 0,Y 439.632,Z 452.974,A -85,B 0,C 180,E1 -9268.168,E2 -9268.168} C_VEL
LIN {X 0,Y 439.761,Z 452.96,A -85,B 0,C 180,E1 -9270,E2 -9270} C_VEL
LIN {X 0,Y 439.618,Z 452.974,A -85,B 0,C 180,E1 -9270.999,E2 -9270.999} C_VEL
LIN {X 0,Y 438.903,Z 453.065,A -85,B 0,C 180,E1 -9271.763,E2 -9271.763} C_VEL
LIN {X 0,Y 435.925,Z 453.435,A -85,B 0,C 180,E1 -9273.002,E2 -9273.002} C_VEL
LIN {X 0,Y 433.473,Z 453.742,A -85,B 0,C 180,E1 -9274.003,E2 -9274.003} C_VEL
LIN {X 0,Y 432.5,Z 453.86,A -85,B 0,C 180,E1 -9274.777,E2 -9274.777} C_VEL
LIN {X 0,Y 432.464,Z 453.864,A -85,B 0,C 180,E1 -9275.039,E2 -9275.039} C_VEL
LIN {X 0,Y 432.583,Z 453.85,A -85,B 0,C 180,E1 -9277.679,E2 -9277.679} C_VEL
LIN {X 0,Y 432.404,Z 453.874,A -85,B 0,C 180,E1 -9281.247,E2 -9281.247} C_VEL
LIN {X 0,Y 432.428,Z 453.869,A -85,B 0,C 180,E1 -9283.152,E2 -9283.152} C_VEL
LIN {X 0,Y 432.409,Z 453.875,A -85,B 0,C 180,E1 -9286.479,E2 -9286.479} C_VEL
LIN {X 0,Y 432.334,Z 453.882,A -85,B 0,C 180,E1 -9289.96,E2 -9289.96} C_VEL
LIN {X 0,Y 432.314,Z 453.885,A -85,B 0,C 180,E1 -9292.964,E2 -9292.964} C_VEL
LIN {X 0,Y 432.359,Z 453.879,A -85,B 0,C 180,E1 -9296.032,E2 -9296.032} C_VEL
LIN {X 0,Y 432.338,Z 453.882,A -85,B 0,C 180,E1 -9299.187,E2 -9299.187} C_VEL
LIN {X 0,Y 432.317,Z 453.885,A -85,B 0,C 180,E1 -9302.443,E2 -9302.443} C_VEL
LIN {X 0,Y 432.339,Z 453.878,A -85,B 0,C 180,E1 -9305.632,E2 -9305.632} C_VEL
LIN {X 0,Y 432.353,Z 453.881,A -85,B 0,C 180,E1 -9308.717,E2 -9308.717} C_VEL
LIN {X 0,Y 432.359,Z 453.877,A -85,B 0,C 180,E1 -9311.793,E2 -9311.793} C_VEL
LIN {X 0,Y 432.371,Z 453.876,A -85,B 0,C 180,E1 -9315.658,E2 -9315.658} C_VEL
LIN {X 0,Y 432.366,Z 453.879,A -85,B 0,C 180,E1 -9318.392,E2 -9318.392} C_VEL
LIN {X 0,Y 432.345,Z 453.879,A -85,B 0,C 180,E1 -9321.852,E2 -9321.852} C_VEL
LIN {X 0,Y 432.332,Z 453.849,A -85,B 0,C 180,E1 -9325.323,E2 -9325.323} C_VEL
LIN {X 0,Y 432.315,Z 453.88,A -85,B 0,C 180,E1 -9328.654,E2 -9328.654} C_VEL
LIN {X 0,Y 432.372,Z 453.861,A -85,B 0,C 180,E1 -9331.369,E2 -9331.369} C_VEL
LIN {X 0,Y 432.355,Z 453.844,A -85,B 0,C 180,E1 -9333.967,E2 -9333.967} C_VEL
LIN {X 0,Y 432.31,Z 453.885,A -85,B 0,C 180,E1 -9337.036,E2 -9337.036} C_VEL
LIN {X 0,Y 432.378,Z 453.868,A -85,B 0,C 180,E1 -9340.515,E2 -9340.515} C_VEL
LIN {X 0,Y 432.421,Z 453.856,A -85,B 0,C 180,E1 -9343.961,E2 -9343.961} C_VEL
LIN {X 0,Y 432.45,Z 453.857,A -85,B 0,C 180,E1 -9347.803,E2 -9347.803} C_VEL
LIN {X 0,Y 432.483,Z 453.861,A -85,B 0,C 180,E1 -9351.59,E2 -9351.59} C_VEL
LIN {X 0,Y 432.592,Z 453.839,A -85,B 0,C 180,E1 -9354.406,E2 -9354.406} C_VEL
LIN {X 0,Y 432.597,Z 453.834,A -85,B 0,C 180,E1 -9358.138,E2 -9358.138} C_VEL
LIN {X 0,Y 432.724,Z 453.832,A -85,B 0,C 180,E1 -9360,E2 -9360} C_VEL
LIN {X 0,Y 432.597,Z 453.842,A -85,B 0,C 180,E1 -9362.794,E2 -9362.794} C_VEL
LIN {X 0,Y 432.563,Z 453.849,A -85,B 0,C 180,E1 -9366.531,E2 -9366.531} C_VEL
LIN {X 0,Y 432.435,Z 453.857,A -85,B 0,C 180,E1 -9369.353,E2 -9369.353} C_VEL
LIN {X 0,Y 432.422,Z 453.859,A -85,B 0,C 180,E1 -9372.804,E2 -9372.804} C_VEL
LIN {X 0,Y 432.404,Z 453.867,A -85,B 0,C 180,E1 -9376.479,E2 -9376.479} C_VEL
LIN {X 0,Y 432.329,Z 453.839,A -85,B 0,C 180,E1 -9379.961,E2 -9379.961} C_VEL
LIN {X 0,Y 432.311,Z 453.877,A -85,B 0,C 180,E1 -9382.965,E2 -9382.965} C_VEL
LIN {X 0,Y 432.357,Z 453.867,A -85,B 0,C 180,E1 -9386.033,E2 -9386.033} C_VEL
LIN {X 0,Y 432.345,Z 453.849,A -85,B 0,C 180,E1 -9389.187,E2 -9389.187} C_VEL
LIN {X 0,Y 432.325,Z 453.883,A -85,B 0,C 180,E1 -9392.295,E2 -9392.295} C_VEL
LIN {X 0,Y 432.334,Z 453.857,A -85,B 0,C 180,E1 -9394.678,E2 -9394.678} C_VEL
LIN {X 0,Y 432.346,Z 453.879,A -85,B 0,C 180,E1 -9398.149,E2 -9398.149} C_VEL
LIN {X 0,Y 432.366,Z 453.874,A -85,B 0,C 180,E1 -9401.608,E2 -9401.608} C_VEL
LIN {X 0,Y 432.373,Z 453.863,A -85,B 0,C 180,E1 -9404.342,E2 -9404.342} C_VEL
LIN {X 0,Y 432.328,Z 453.873,A -85,B 0,C 180,E1 -9408.203,E2 -9408.203} C_VEL
LIN {X 0,Y 432.341,Z 453.983,A -85,B 0,C 180,E1 -9411.285,E2 -9411.285} C_VEL
LIN {X 0,Y 433.011,Z 456.528,A -85,B 0,C 180,E1 -9411.921,E2 -9411.921} C_VEL
LIN {X 0,Y 436.861,Z 470.516,A -85,B 0,C 180,E1 -9414.951,E2 -9414.951} C_VEL
LIN {X 0,Y 439.494,Z 480.925,A -85,B 0,C 180,E1 -9417.031,E2 -9417.031} C_VEL
LIN {X 0,Y 442.602,Z 488.175,A -85,B 0,C 180,E1 -9417.452,E2 -9417.452} C_VEL
LIN {X 0,Y 450.245,Z 518.895,A -85,B 0,C 180,E1 -9418.628,E2 -9418.628} C_VEL
LIN {X 0,Y 447.215,Z 677.009,A -85,B 0,C 180,E1 -9421.264,E2 -9421.264} C_VEL
LIN {X 0,Y 446.597,Z 700.045,A -85,B 0,C 180,E1 -9421.702,E2 -9421.702} C_VEL
LIN {X 0,Y 445.689,Z 716.239,A -85,B 0,C 180,E1 -9422.191,E2 -9422.191} C_VEL
LIN {X 0,Y 444.779,Z 729.699,A -85,B 0,C 180,E1 -9422.728,E2 -9422.728} C_VEL
LIN {X 0,Y 443.786,Z 742.511,A -85,B 0,C 180,E1 -9423.362,E2 -9423.362} C_VEL
LIN {X 0,Y 442.641,Z 755.153,A -85,B 0,C 180,E1 -9424.112,E2 -9424.112} C_VEL
LIN {X 0,Y 441.375,Z 768.042,A -85,B 0,C 180,E1 -9425.021,E2 -9425.021} C_VEL
LIN {X 0,Y 440.17,Z 779.637,A -85,B 0,C 180,E1 -9425.975,E2 -9425.975} C_VEL
LIN {X 0,Y 438.874,Z 790.777,A -85,B 0,C 180,E1 -9427.025,E2 -9427.025} C_VEL
LIN {X 0,Y 437.621,Z 801.623,A -85,B 0,C 180,E1 -9428.2,E2 -9428.2} C_VEL
LIN {X 0,Y 436.663,Z 810.314,A -85,B 0,C 180,E1 -9429.263,E2 -9429.263} C_VEL
LIN {X 0,Y 435.481,Z 820.527,A -85,B 0,C 180,E1 -9430.681,E2 -9430.681} C_VEL
LIN {X 0,Y 434.448,Z 829.487,A -85,B 0,C 180,E1 -9432.1,E2 -9432.1} C_VEL
LIN {X 0,Y 433.723,Z 837.384,A -85,B 0,C 180,E1 -9433.527,E2 -9433.527} C_VEL
LIN {X 0,Y 432.984,Z 844.346,A -85,B 0,C 180,E1 -9434.948,E2 -9434.948} C_VEL
LIN {X 0,Y 432.493,Z 850.487,A -85,B 0,C 180,E1 -9436.372,E2 -9436.372} C_VEL
LIN {X 0,Y 431.945,Z 857.428,A -85,B 0,C 180,E1 -9438.265,E2 -9438.265} C_VEL
LIN {X 0,Y 431.524,Z 863.176,A -85,B 0,C 180,E1 -9440.154,E2 -9440.154} C_VEL
LIN {X 0,Y 431.4,Z 866.784,A -85,B 0,C 180,E1 -9441.569,E2 -9441.569} C_VEL
LIN {X 0,Y 431.319,Z 871.034,A -85,B 0,C 180,E1 -9443.69,E2 -9443.69} C_VEL
LIN {X 0,Y 431.209,Z 873.465,A -85,B 0,C 180,E1 -9445.326,E2 -9445.326} C_VEL
LIN {X 0,Y 431.208,Z 875.34,A -85,B 0,C 180,E1 -9447.197,E2 -9447.197} C_VEL
LIN {X 0,Y 431.192,Z 876.012,A -85,B 0,C 180,E1 -9448.132,E2 -9448.132} C_VEL
LIN {X 0,Y 431.118,Z 876.48,A -85,B 0,C 180,E1 -9450,E2 -9450} C_VEL
LIN {X 0,Y 431.192,Z 876.012,A -85,B 0,C 180,E1 -9451.868,E2 -9451.868} C_VEL
LIN {X 0,Y 431.142,Z 874.594,A -85,B 0,C 180,E1 -9453.738,E2 -9453.738} C_VEL
LIN {X 0,Y 431.223,Z 872.22,A -85,B 0,C 180,E1 -9455.612,E2 -9455.612} C_VEL
LIN {X 0,Y 431.371,Z 868.859,A -85,B 0,C 180,E1 -9457.489,E2 -9457.489} C_VEL
LIN {X 0,Y 431.489,Z 864.461,A -85,B 0,C 180,E1 -9459.374,E2 -9459.374} C_VEL
LIN {X 0,Y 431.82,Z 858.971,A -85,B 0,C 180,E1 -9461.262,E2 -9461.262} C_VEL
LIN {X 0,Y 432.148,Z 854.285,A -85,B 0,C 180,E1 -9462.638,E2 -9462.638} C_VEL
LIN {X 0,Y 432.833,Z 846.453,A -85,B 0,C 180,E1 -9464.576,E2 -9464.576} C_VEL
LIN {X 0,Y 433.498,Z 839.803,A -85,B 0,C 180,E1 -9465.998,E2 -9465.998} C_VEL
LIN {X 0,Y 434.211,Z 832.209,A -85,B 0,C 180,E1 -9467.43,E2 -9467.43} C_VEL
LIN {X 0,Y 435.099,Z 823.659,A -85,B 0,C 180,E1 -9468.847,E2 -9468.847} C_VEL
LIN {X 0,Y 436.233,Z 813.866,A -85,B 0,C 180,E1 -9470.266,E2 -9470.266} C_VEL
LIN {X 0,Y 437.318,Z 804.382,A -85,B 0,C 180,E1 -9471.477,E2 -9471.477} C_VEL
LIN {X 0,Y 438.624,Z 793.066,A -85,B 0,C 180,E1 -9472.739,E2 -9472.739} C_VEL
LIN {X 0,Y 439.855,Z 782.248,A -85,B 0,C 180,E1 -9473.793,E2 -9473.793} C_VEL
LIN {X 0,Y 441.02,Z 771.35,A -85,B 0,C 180,E1 -9474.724,E2 -9474.724} C_VEL
LIN {X 0,Y 442.132,Z 760.38,A -85,B 0,C 180,E1 -9475.541,E2 -9475.541} C_VEL
LIN {X 0,Y 443.306,Z 747.642,A -85,B 0,C 180,E1 -9476.352,E2 -9476.352} C_VEL
LIN {X 0,Y 444.407,Z 734.639,A -85,B 0,C 180,E1 -9477.042,E2 -9477.042} C_VEL
LIN {X 0,Y 445.401,Z 720.877,A -85,B 0,C 180,E1 -9477.636,E2 -9477.636} C_VEL
LIN {X 0,Y 446.18,Z 708.622,A -85,B 0,C 180,E1 -9478.053,E2 -9478.053} C_VEL
LIN {X 0,Y 446.796,Z 694.593,A -85,B 0,C 180,E1 -9478.412,E2 -9478.412} C_VEL
LIN {X 0,Y 447.599,Z 657.307,A -85,B 0,C 180,E1 -9479.062,E2 -9479.062} C_VEL
LIN {X 0,Y 450.238,Z 519.578,A -85,B 0,C 180,E1 -9481.36,E2 -9481.36} C_VEL
LIN {X 0,Y 445.951,Z 501.128,A -85,B 0,C 180,E1 -9482.035,E2 -9482.035} C_VEL
LIN {X 0,Y 442.171,Z 486.992,A -85,B 0,C 180,E1 -9482.606,E2 -9482.606} C_VEL
LIN {X 0,Y 439.429,Z 480.808,A -85,B 0,C 180,E1 -9482.986,E2 -9482.986} C_VEL
LIN {X 0,Y 436.073,Z 467.516,A -85,B 0,C 180,E1 -9485.676,E2 -9485.676} C_VEL
LIN {X 0,Y 432.42,Z 454.423,A -85,B 0,C 180,E1 -9488.555,E2 -9488.555} C_VEL
LIN {X 0,Y 432.317,Z 453.882,A -85,B 0,C 180,E1 -9488.811,E2 -9488.811} C_VEL
LIN {X 0,Y 432.328,Z 453.873,A -85,B 0,C 180,E1 -9491.797,E2 -9491.797} C_VEL
LIN {X 0,Y 432.373,Z 453.863,A -85,B 0,C 180,E1 -9495.658,E2 -9495.658} C_VEL
LIN {X 0,Y 432.366,Z 453.874,A -85,B 0,C 180,E1 -9498.392,E2 -9498.392} C_VEL
LIN {X 0,Y 432.346,Z 453.879,A -85,B 0,C 180,E1 -9501.851,E2 -9501.851} C_VEL
LIN {X 0,Y 432.334,Z 453.857,A -85,B 0,C 180,E1 -9505.322,E2 -9505.322} C_VEL
LIN {X 0,Y 432.323,Z 453.879,A -85,B 0,C 180,E1 -9508.654,E2 -9508.654} C_VEL
LIN {X 0,Y 432.377,Z 453.84,A -85,B 0,C 180,E1 -9511.876,E2 -9511.876} C_VEL
LIN {X 0,Y 432.344,Z 453.877,A -85,B 0,C 180,E1 -9514.998,E2 -9514.998} C_VEL
LIN {X 0,Y 432.349,Z 453.855,A -85,B 0,C 180,E1 -9518.045,E2 -9518.045} C_VEL
LIN {X 0,Y 432.378,Z 453.842,A -85,B 0,C 180,E1 -9521.029,E2 -9521.029} C_VEL
LIN {X 0,Y 432.422,Z 453.868,A -85,B 0,C 180,E1 -9523.961,E2 -9523.961} C_VEL
LIN {X 0,Y 432.451,Z 453.859,A -85,B 0,C 180,E1 -9527.803,E2 -9527.803} C_VEL
LIN {X 0,Y 432.483,Z 453.848,A -85,B 0,C 180,E1 -9531.59,E2 -9531.59} C_VEL
LIN {X 0,Y 432.589,Z 453.851,A -85,B 0,C 180,E1 -9534.406,E2 -9534.406} C_VEL
LIN {X 0,Y 432.597,Z 453.845,A -85,B 0,C 180,E1 -9538.138,E2 -9538.138} C_VEL
LIN {X 0,Y 432.724,Z 453.831,A -85,B 0,C 180,E1 -9540,E2 -9540} C_VEL
LIN {X 0,Y 432.597,Z 453.845,A -85,B 0,C 180,E1 -9542.793,E2 -9542.793} C_VEL
LIN {X 0,Y 432.565,Z 453.84,A -85,B 0,C 180,E1 -9546.53,E2 -9546.53} C_VEL
LIN {X 0,Y 432.435,Z 453.863,A -85,B 0,C 180,E1 -9549.353,E2 -9549.353} C_VEL
LIN {X 0,Y 432.421,Z 453.869,A -85,B 0,C 180,E1 -9552.803,E2 -9552.803} C_VEL
LIN {X 0,Y 432.403,Z 453.862,A -85,B 0,C 180,E1 -9556.479,E2 -9556.479} C_VEL
LIN {X 0,Y 432.33,Z 453.874,A -85,B 0,C 180,E1 -9559.961,E2 -9559.961} C_VEL
LIN {X 0,Y 432.31,Z 453.885,A -85,B 0,C 180,E1 -9562.964,E2 -9562.964} C_VEL
LIN {X 0,Y 432.355,Z 453.844,A -85,B 0,C 180,E1 -9566.033,E2 -9566.033} C_VEL
LIN {X 0,Y 432.344,Z 453.873,A -85,B 0,C 180,E1 -9569.187,E2 -9569.187} C_VEL
LIN {X 0,Y 432.317,Z 453.872,A -85,B 0,C 180,E1 -9572.294,E2 -9572.294} C_VEL
LIN {X 0,Y 432.332,Z 453.849,A -85,B 0,C 180,E1 -9574.677,E2 -9574.677} C_VEL
LIN {X 0,Y 432.346,Z 453.879,A -85,B 0,C 180,E1 -9578.148,E2 -9578.148} C_VEL
LIN {X 0,Y 432.366,Z 453.879,A -85,B 0,C 180,E1 -9581.608,E2 -9581.608} C_VEL
LIN {X 0,Y 432.371,Z 453.876,A -85,B 0,C 180,E1 -9584.342,E2 -9584.342} C_VEL
LIN {X 0,Y 432.36,Z 453.877,A -85,B 0,C 180,E1 -9588.393,E2 -9588.393} C_VEL
LIN {X 0,Y 432.345,Z 453.882,A -85,B 0,C 180,E1 -9591.852,E2 -9591.852} C_VEL
LIN {X 0,Y 432.335,Z 453.884,A -85,B 0,C 180,E1 -9595.323,E2 -9595.323} C_VEL
LIN {X 0,Y 432.316,Z 453.883,A -85,B 0,C 180,E1 -9598.654,E2 -9598.654} C_VEL
LIN {X 0,Y 432.378,Z 453.878,A -85,B 0,C 180,E1 -9601.877,E2 -9601.877} C_VEL
LIN {X 0,Y 432.347,Z 453.88,A -85,B 0,C 180,E1 -9604.999,E2 -9604.999} C_VEL
LIN {X 0,Y 432.354,Z 453.88,A -85,B 0,C 180,E1 -9608.046,E2 -9608.046} C_VEL
LIN {X 0,Y 432.382,Z 453.877,A -85,B 0,C 180,E1 -9611.03,E2 -9611.03} C_VEL
LIN {X 0,Y 432.427,Z 453.871,A -85,B 0,C 180,E1 -9613.961,E2 -9613.961} C_VEL
LIN {X 0,Y 432.477,Z 453.866,A -85,B 0,C 180,E1 -9617.804,E2 -9617.804} C_VEL
LIN {X 0,Y 432.489,Z 453.864,A -85,B 0,C 180,E1 -9621.59,E2 -9621.59} C_VEL
LIN {X 0,Y 432.594,Z 453.852,A -85,B 0,C 180,E1 -9624.406,E2 -9624.406} C_VEL
LIN {X 0,Y 432.603,Z 453.849,A -85,B 0,C 180,E1 -9628.138,E2 -9628.138} C_VEL
LIN {X 0,Y 432.73,Z 453.836,A -85,B 0,C 180,E1 -9630,E2 -9630} C_VEL
LIN {X 0,Y 432.602,Z 453.85,A -85,B 0,C 180,E1 -9632.793,E2 -9632.793} C_VEL
LIN {X 0,Y 432.464,Z 453.864,A -85,B 0,C 180,E1 -9635.039,E2 -9635.039} C_VEL
LIN {X 0,Y 431.904,Z 453.937,A -85,B 0,C 180,E1 -9635.818,E2 -9635.818} C_VEL
LIN {X 0,Y 429.056,Z 454.291,A -85,B 0,C 180,E1 -9637.083,E2 -9637.083} C_VEL
LIN {X 0,Y 426.571,Z 454.601,A -85,B 0,C 180,E1 -9638.104,E2 -9638.104} C_VEL
LIN {X 0,Y 425.491,Z 454.733,A -85,B 0,C 180,E1 -9638.894,E2 -9638.894} C_VEL
LIN {X 0,Y 425.4,Z 454.744,A -85,B 0,C 180,E1 -9639.162,E2 -9639.162} C_VEL
LIN {X 0,Y 425.4,Z 454.745,A -85,B 0,C 180,E1 -9642.91,E2 -9642.91} C_VEL
LIN {X 0,Y 425.357,Z 454.752,A -85,B 0,C 180,E1 -9646.605,E2 -9646.605} C_VEL
LIN {X 0,Y 425.324,Z 454.756,A -85,B 0,C 180,E1 -9649.635,E2 -9649.635} C_VEL
LIN {X 0,Y 425.302,Z 454.759,A -85,B 0,C 180,E1 -9653.365,E2 -9653.365} C_VEL
LIN {X 0,Y 425.344,Z 454.753,A -85,B 0,C 180,E1 -9656.844,E2 -9656.844} C_VEL
LIN {X 0,Y 425.285,Z 454.759,A -85,B 0,C 180,E1 -9659.719,E2 -9659.719} C_VEL
LIN {X 0,Y 425.276,Z 454.762,A -85,B 0,C 180,E1 -9663.048,E2 -9663.048} C_VEL
LIN {X 0,Y 425.279,Z 454.759,A -85,B 0,C 180,E1 -9665.929,E2 -9665.929} C_VEL
LIN {X 0,Y 425.306,Z 454.759,A -85,B 0,C 180,E1 -9669.045,E2 -9669.045} C_VEL
LIN {X 0,Y 425.308,Z 454.756,A -85,B 0,C 180,E1 -9671.962,E2 -9671.962} C_VEL
LIN {X 0,Y 425.306,Z 454.758,A -85,B 0,C 180,E1 -9675.279,E2 -9675.279} C_VEL
LIN {X 0,Y 425.303,Z 454.76,A -85,B 0,C 180,E1 -9678.625,E2 -9678.625} C_VEL
LIN {X 0,Y 425.317,Z 454.758,A -85,B 0,C 180,E1 -9681.104,E2 -9681.104} C_VEL
LIN {X 0,Y 425.292,Z 454.735,A -85,B 0,C 180,E1 -9684.664,E2 -9684.664} C_VEL
LIN {X 0,Y 425.258,Z 454.755,A -85,B 0,C 180,E1 -9688.073,E2 -9688.073} C_VEL
LIN {X 0,Y 425.329,Z 454.737,A -85,B 0,C 180,E1 -9691.368,E2 -9691.368} C_VEL
LIN {X 0,Y 425.286,Z 454.73,A -85,B 0,C 180,E1 -9694.555,E2 -9694.555} C_VEL
LIN {X 0,Y 425.279,Z 454.759,A -85,B 0,C 180,E1 -9697.661,E2 -9697.661} C_VEL
LIN {X 0,Y 425.353,Z 454.744,A -85,B 0,C 180,E1 -9700.704,E2 -9700.704} C_VEL
LIN {X 0,Y 425.379,Z 454.735,A -85,B 0,C 180,E1 -9703.688,E2 -9703.688} C_VEL
LIN {X 0,Y 425.403,Z 454.737,A -85,B 0,C 180,E1 -9707.598,E2 -9707.598} C_VEL
LIN {X 0,Y 425.434,Z 454.741,A -85,B 0,C 180,E1 -9711.45,E2 -9711.45} C_VEL
LIN {X 0,Y 425.548,Z 454.717,A -85,B 0,C 180,E1 -9714.313,E2 -9714.313} C_VEL
LIN {X 0,Y 425.566,Z 454.71,A -85,B 0,C 180,E1 -9718.107,E2 -9718.107} C_VEL
LIN {X 0,Y 425.694,Z 454.708,A -85,B 0,C 180,E1 -9720,E2 -9720} C_VEL
LIN {X 0,Y 425.549,Z 454.72,A -85,B 0,C 180,E1 -9722.84,E2 -9722.84} C_VEL
LIN {X 0,Y 425.565,Z 454.726,A -85,B 0,C 180,E1 -9725.687,E2 -9725.687} C_VEL
LIN {X 0,Y 425.434,Z 454.725,A -85,B 0,C 180,E1 -9728.55,E2 -9728.55} C_VEL
LIN {X 0,Y 425.404,Z 454.734,A -85,B 0,C 180,E1 -9732.402,E2 -9732.402} C_VEL
LIN {X 0,Y 425.38,Z 454.743,A -85,B 0,C 180,E1 -9736.312,E2 -9736.312} C_VEL
LIN {X 0,Y 425.32,Z 454.711,A -85,B 0,C 180,E1 -9739.636,E2 -9739.636} C_VEL
LIN {X 0,Y 425.28,Z 454.743,A -85,B 0,C 180,E1 -9742.339,E2 -9742.339} C_VEL
LIN {X 0,Y 425.289,Z 454.758,A -85,B 0,C 180,E1 -9745.446,E2 -9745.446} C_VEL
LIN {X 0,Y 425.331,Z 454.716,A -85,B 0,C 180,E1 -9748.632,E2 -9748.632} C_VEL
LIN {X 0,Y 425.266,Z 454.764,A -85,B 0,C 180,E1 -9751.927,E2 -9751.927} C_VEL
LIN {X 0,Y 425.294,Z 454.734,A -85,B 0,C 180,E1 -9755.336,E2 -9755.336} C_VEL
LIN {X 0,Y 425.306,Z 454.747,A -85,B 0,C 180,E1 -9759.046,E2 -9759.046} C_VEL
LIN {X 0,Y 425.326,Z 454.753,A -85,B 0,C 180,E1 -9762.647,E2 -9762.647} C_VEL
LIN {X 0,Y 425.292,Z 454.753,A -85,B 0,C 180,E1 -9765.282,E2 -9765.282} C_VEL
LIN {X 0,Y 425.269,Z 454.757,A -85,B 0,C 180,E1 -9768.622,E2 -9768.622} C_VEL
LIN {X 0,Y 425.285,Z 454.852,A -85,B 0,C 180,E1 -9770.752,E2 -9770.752} C_VEL
LIN {X 0,Y 426.235,Z 458.156,A -85,B 0,C 180,E1 -9771.584,E2 -9771.584} C_VEL
LIN {X 0,Y 430.163,Z 472.621,A -85,B 0,C 180,E1 -9774.775,E2 -9774.775} C_VEL
LIN {X 0,Y 432.14,Z 480.629,A -85,B 0,C 180,E1 -9776.396,E2 -9776.396} C_VEL
LIN {X 0,Y 436.869,Z 490.711,A -85,B 0,C 180,E1 -9777.023,E2 -9777.023} C_VEL
LIN {X 0,Y 444.19,Z 520.341,A -85,B 0,C 180,E1 -9778.181,E2 -9778.181} C_VEL
LIN {X 0,Y 440.71,Z 690.123,A -85,B 0,C 180,E1 -9781.061,E2 -9781.061} C_VEL
LIN {X 0,Y 440.021,Z 704.53,A -85,B 0,C 180,E1 -9781.393,E2 -9781.393} C_VEL
LIN {X 0,Y 439.262,Z 717.897,A -85,B 0,C 180,E1 -9781.827,E2 -9781.827} C_VEL
LIN {X 0,Y 438.336,Z 730.723,A -85,B 0,C 180,E1 -9782.357,E2 -9782.357} C_VEL
LIN {X 0,Y 437.316,Z 743.326,A -85,B 0,C 180,E1 -9783,E2 -9783} C_VEL
LIN {X 0,Y 436.213,Z 754.942,A -85,B 0,C 180,E1 -9783.701,E2 -9783.701} C_VEL
LIN {X 0,Y 435.025,Z 766.593,A -85,B 0,C 180,E1 -9784.525,E2 -9784.525} C_VEL
LIN {X 0,Y 433.593,Z 779.424,A -85,B 0,C 180,E1 -9785.587,E2 -9785.587} C_VEL
LIN {X 0,Y 432.204,Z 790.562,A -85,B 0,C 180,E1 -9786.65,E2 -9786.65} C_VEL
LIN {X 0,Y 430.972,Z 801.412,A -85,B 0,C 180,E1 -9787.846,E2 -9787.846} C_VEL
LIN {X 0,Y 429.715,Z 811.878,A -85,B 0,C 180,E1 -9789.163,E2 -9789.163} C_VEL
LIN {X 0,Y 428.664,Z 820.313,A -85,B 0,C 180,E1 -9790.361,E2 -9790.361} C_VEL
LIN {X 0,Y 427.575,Z 829.274,A -85,B 0,C 180,E1 -9791.803,E2 -9791.803} C_VEL
LIN {X 0,Y 426.775,Z 837.17,A -85,B 0,C 180,E1 -9793.251,E2 -9793.251} C_VEL
LIN {X 0,Y 426.01,Z 844.132,A -85,B 0,C 180,E1 -9794.695,E2 -9794.695} C_VEL
LIN {X 0,Y 425.499,Z 850.274,A -85,B 0,C 180,E1 -9796.143,E2 -9796.143} C_VEL
LIN {X 0,Y 424.919,Z 857.216,A -85,B 0,C 180,E1 -9798.069,E2 -9798.069} C_VEL
LIN {X 0,Y 424.465,Z 862.965,A -85,B 0,C 180,E1 -9799.988,E2 -9799.988} C_VEL
LIN {X 0,Y 424.338,Z 866.573,A -85,B 0,C 180,E1 -9801.428,E2 -9801.428} C_VEL
LIN {X 0,Y 424.235,Z 870.416,A -85,B 0,C 180,E1 -9803.341,E2 -9803.341} C_VEL
LIN {X 0,Y 424.135,Z 873.255,A -85,B 0,C 180,E1 -9805.248,E2 -9805.248} C_VEL
LIN {X 0,Y 424.104,Z 875.13,A -85,B 0,C 180,E1 -9807.15,E2 -9807.15} C_VEL
LIN {X 0,Y 424.118,Z 875.803,A -85,B 0,C 180,E1 -9808.101,E2 -9808.101} C_VEL
LIN {X 0,Y 424.037,Z 876.271,A -85,B 0,C 180,E1 -9810,E2 -9810} C_VEL
LIN {X 0,Y 424.118,Z 875.803,A -85,B 0,C 180,E1 -9811.899,E2 -9811.899} C_VEL
LIN {X 0,Y 424.054,Z 874.384,A -85,B 0,C 180,E1 -9813.801,E2 -9813.801} C_VEL
LIN {X 0,Y 424.225,Z 871.049,A -85,B 0,C 180,E1 -9816.281,E2 -9816.281} C_VEL
LIN {X 0,Y 424.283,Z 867.61,A -85,B 0,C 180,E1 -9818.094,E2 -9818.094} C_VEL
LIN {X 0,Y 424.4,Z 864.249,A -85,B 0,C 180,E1 -9819.532,E2 -9819.532} C_VEL
LIN {X 0,Y 424.762,Z 858.758,A -85,B 0,C 180,E1 -9821.452,E2 -9821.452} C_VEL
LIN {X 0,Y 425.168,Z 853.664,A -85,B 0,C 180,E1 -9822.958,E2 -9822.958} C_VEL
LIN {X 0,Y 425.836,Z 846.239,A -85,B 0,C 180,E1 -9824.821,E2 -9824.821} C_VEL
LIN {X 0,Y 426.565,Z 839.59,A -85,B 0,C 180,E1 -9826.265,E2 -9826.265} C_VEL
LIN {X 0,Y 427.316,Z 832.037,A -85,B 0,C 180,E1 -9827.713,E2 -9827.713} C_VEL
LIN {X 0,Y 428.282,Z 823.446,A -85,B 0,C 180,E1 -9829.159,E2 -9829.159} C_VEL
LIN {X 0,Y 429.481,Z 813.653,A -85,B 0,C 180,E1 -9830.598,E2 -9830.598} C_VEL
LIN {X 0,Y 430.609,Z 804.387,A -85,B 0,C 180,E1 -9831.801,E2 -9831.801} C_VEL
LIN {X 0,Y 431.846,Z 793.997,A -85,B 0,C 180,E1 -9832.99,E2 -9832.99} C_VEL
LIN {X 0,Y 433.291,Z 782.036,A -85,B 0,C 180,E1 -9834.176,E2 -9834.176} C_VEL
LIN {X 0,Y 434.618,Z 770.346,A -85,B 0,C 180,E1 -9835.18,E2 -9835.18} C_VEL
LIN {X 0,Y 435.851,Z 758.426,A -85,B 0,C 180,E1 -9836.065,E2 -9836.065} C_VEL
LIN {X 0,Y 437.001,Z 746.404,A -85,B 0,C 180,E1 -9836.827,E2 -9836.827} C_VEL
LIN {X 0,Y 438.06,Z 734.428,A -85,B 0,C 180,E1 -9837.467,E2 -9837.467} C_VEL
LIN {X 0,Y 439.071,Z 721.191,A -85,B 0,C 180,E1 -9838.047,E2 -9838.047} C_VEL
LIN {X 0,Y 439.892,Z 708.118,A -85,B 0,C 180,E1 -9838.499,E2 -9838.499} C_VEL
LIN {X 0,Y 440.559,Z 694.383,A -85,B 0,C 180,E1 -9838.852,E2 -9838.852} C_VEL
LIN {X 0,Y 441.413,Z 657.097,A -85,B 0,C 180,E1 -9839.509,E2 -9839.509} C_VEL
LIN {X 0,Y 444.174,Z 520.354,A -85,B 0,C 180,E1 -9841.82,E2 -9841.82} C_VEL
LIN {X 0,Y 436.976,Z 491.082,A -85,B 0,C 180,E1 -9842.961,E2 -9842.961} C_VEL
LIN {X 0,Y 432.152,Z 480.582,A -85,B 0,C 180,E1 -9843.606,E2 -9843.606} C_VEL
LIN {X 0,Y 429.05,Z 468.354,A -85,B 0,C 180,E1 -9846.134,E2 -9846.134} C_VEL
LIN {X 0,Y 425.33,Z 455.021,A -85,B 0,C 180,E1 -9849.17,E2 -9849.17} C_VEL
LIN {X 0,Y 425.278,Z 454.73,A -85,B 0,C 180,E1 -9849.54,E2 -9849.54} C_VEL
LIN {X 0,Y 425.27,Z 454.751,A -85,B 0,C 180,E1 -9852.652,E2 -9852.652} C_VEL
LIN {X 0,Y 425.314,Z 454.743,A -85,B 0,C 180,E1 -9856.051,E2 -9856.051} C_VEL
LIN {X 0,Y 425.303,Z 454.753,A -85,B 0,C 180,E1 -9858.625,E2 -9858.625} C_VEL
LIN {X 0,Y 425.317,Z 454.746,A -85,B 0,C 180,E1 -9861.103,E2 -9861.103} C_VEL
LIN {X 0,Y 425.294,Z 454.734,A -85,B 0,C 180,E1 -9864.664,E2 -9864.664} C_VEL
LIN {X 0,Y 425.266,Z 454.764,A -85,B 0,C 180,E1 -9868.073,E2 -9868.073} C_VEL
LIN {X 0,Y 425.331,Z 454.716,A -85,B 0,C 180,E1 -9871.368,E2 -9871.368} C_VEL
LIN {X 0,Y 425.289,Z 454.758,A -85,B 0,C 180,E1 -9874.554,E2 -9874.554} C_VEL
LIN {X 0,Y 425.28,Z 454.743,A -85,B 0,C 180,E1 -9877.661,E2 -9877.661} C_VEL
LIN {X 0,Y 425.354,Z 454.71,A -85,B 0,C 180,E1 -9880.704,E2 -9880.704} C_VEL
LIN {X 0,Y 425.38,Z 454.742,A -85,B 0,C 180,E1 -9883.688,E2 -9883.688} C_VEL
LIN {X 0,Y 425.404,Z 454.735,A -85,B 0,C 180,E1 -9887.598,E2 -9887.598} C_VEL
LIN {X 0,Y 425.434,Z 454.725,A -85,B 0,C 180,E1 -9891.45,E2 -9891.45} C_VEL
LIN {X 0,Y 425.565,Z 454.727,A -85,B 0,C 180,E1 -9894.313,E2 -9894.313} C_VEL
LIN {X 0,Y 425.566,Z 454.72,A -85,B 0,C 180,E1 -9898.107,E2 -9898.107} C_VEL
LIN {X 0,Y 425.694,Z 454.707,A -85,B 0,C 180,E1 -9900,E2 -9900} C_VEL
LIN {X 0,Y 425.549,Z 454.723,A -85,B 0,C 180,E1 -9902.84,E2 -9902.84} C_VEL
LIN {X 0,Y 425.522,Z 454.717,A -85,B 0,C 180,E1 -9906.639,E2 -9906.639} C_VEL
LIN {X 0,Y 425.393,Z 454.739,A -85,B 0,C 180,E1 -9909.509,E2 -9909.509} C_VEL
LIN {X 0,Y 425.384,Z 454.747,A -85,B 0,C 180,E1 -9912.904,E2 -9912.904} C_VEL
LIN {X 0,Y 425.352,Z 454.741,A -85,B 0,C 180,E1 -9916.605,E2 -9916.605} C_VEL
LIN {X 0,Y 425.319,Z 454.747,A -85,B 0,C 180,E1 -9919.636,E2 -9919.636} C_VEL
LIN {X 0,Y 425.279,Z 454.759,A -85,B 0,C 180,E1 -9922.339,E2 -9922.339} C_VEL
LIN {X 0,Y 425.286,Z 454.73,A -85,B 0,C 180,E1 -9925.445,E2 -9925.445} C_VEL
LIN {X 0,Y 425.329,Z 454.737,A -85,B 0,C 180,E1 -9928.632,E2 -9928.632} C_VEL
LIN {X 0,Y 425.258,Z 454.755,A -85,B 0,C 180,E1 -9931.927,E2 -9931.927} C_VEL
LIN {X 0,Y 425.292,Z 454.735,A -85,B 0,C 180,E1 -9935.336,E2 -9935.336} C_VEL
LIN {X 0,Y 425.306,Z 454.76,A -85,B 0,C 180,E1 -9939.046,E2 -9939.046} C_VEL
LIN {X 0,Y 425.324,Z 454.755,A -85,B 0,C 180,E1 -9942.646,E2 -9942.646} C_VEL
LIN {X 0,Y 425.287,Z 454.761,A -85,B 0,C 180,E1 -9945.282,E2 -9945.282} C_VEL
LIN {X 0,Y 425.297,Z 454.757,A -85,B 0,C 180,E1 -9948.625,E2 -9948.625} C_VEL
LIN {X 0,Y 425.316,Z 454.758,A -85,B 0,C 180,E1 -9951.104,E2 -9951.104} C_VEL
LIN {X 0,Y 425.294,Z 454.757,A -85,B 0,C 180,E1 -9954.665,E2 -9954.665} C_VEL
LIN {X 0,Y 425.259,Z 454.763,A -85,B 0,C 180,E1 -9958.073,E2 -9958.073} C_VEL
LIN {X 0,Y 425.326,Z 454.755,A -85,B 0,C 180,E1 -9961.368,E2 -9961.368} C_VEL
LIN {X 0,Y 425.291,Z 454.758,A -85,B 0,C 180,E1 -9964.555,E2 -9964.555} C_VEL
LIN {X 0,Y 425.283,Z 454.762,A -85,B 0,C 180,E1 -9967.662,E2 -9967.662} C_VEL
LIN {X 0,Y 425.358,Z 454.752,A -85,B 0,C 180,E1 -9970.704,E2 -9970.704} C_VEL
LIN {X 0,Y 425.384,Z 454.749,A -85,B 0,C 180,E1 -9973.689,E2 -9973.689} C_VEL
LIN {X 0,Y 425.426,Z 454.745,A -85,B 0,C 180,E1 -9977.599,E2 -9977.599} C_VEL
LIN {X 0,Y 425.439,Z 454.741,A -85,B 0,C 180,E1 -9981.45,E2 -9981.45} C_VEL
LIN {X 0,Y 425.551,Z 454.729,A -85,B 0,C 180,E1 -9984.313,E2 -9984.313} C_VEL
LIN {X 0,Y 425.572,Z 454.724,A -85,B 0,C 180,E1 -9988.107,E2 -9988.107} C_VEL
LIN {X 0,Y 425.7,Z 454.711,A -85,B 0,C 180,E1 -9990,E2 -9990} C_VEL
LIN {X 0,Y 425.554,Z 454.728,A -85,B 0,C 180,E1 -9992.84,E2 -9992.84} C_VEL
LIN {X 0,Y 425.527,Z 454.731,A -85,B 0,C 180,E1 -9996.639,E2 -9996.639} C_VEL
LIN {X 0,Y 425.4,Z 454.744,A -85,B 0,C 180,E1 -9999.162,E2 -9999.162} C_VEL
LIN {X 0,Y 424.73,Z 454.831,A -85,B 0,C 180,E1 -9999.951,E2 -9999.951} C_VEL
LIN {X 0,Y 421.884,Z 455.185,A -85,B 0,C 180,E1 -10001.235,E2 -10001.235} C_VEL
LIN {X 0,Y 419.47,Z 455.487,A -85,B 0,C 180,E1 -10002.271,E2 -10002.271} C_VEL
LIN {X 0,Y 418.421,Z 455.614,A -85,B 0,C 180,E1 -10003.072,E2 -10003.072} C_VEL
LIN {X 0,Y 418.329,Z 455.626,A -85,B 0,C 180,E1 -10003.344,E2 -10003.344} C_VEL
LIN {X 0,Y 418.309,Z 455.629,A -85,B 0,C 180,E1 -10006.735,E2 -10006.735} C_VEL
LIN {X 0,Y 418.266,Z 455.634,A -85,B 0,C 180,E1 -10009.79,E2 -10009.79} C_VEL
LIN {X 0,Y 418.233,Z 455.638,A -85,B 0,C 180,E1 -10012.736,E2 -10012.736} C_VEL
LIN {X 0,Y 418.266,Z 455.634,A -85,B 0,C 180,E1 -10015.904,E2 -10015.904} C_VEL
LIN {X 0,Y 418.259,Z 455.636,A -85,B 0,C 180,E1 -10019.162,E2 -10019.162} C_VEL
LIN {X 0,Y 418.252,Z 455.636,A -85,B 0,C 180,E1 -10022.844,E2 -10022.844} C_VEL
LIN {X 0,Y 418.243,Z 455.638,A -85,B 0,C 180,E1 -10026.238,E2 -10026.238} C_VEL
LIN {X 0,Y 418.258,Z 455.634,A -85,B 0,C 180,E1 -10029.68,E2 -10029.68} C_VEL
LIN {X 0,Y 418.238,Z 455.639,A -85,B 0,C 180,E1 -10032.323,E2 -10032.323} C_VEL
LIN {X 0,Y 418.251,Z 455.638,A -85,B 0,C 180,E1 -10035.112,E2 -10035.112} C_VEL
LIN {X 0,Y 418.285,Z 455.631,A -85,B 0,C 180,E1 -10037.773,E2 -10037.773} C_VEL
LIN {X 0,Y 418.259,Z 455.635,A -85,B 0,C 180,E1 -10041.559,E2 -10041.559} C_VEL
LIN {X 0,Y 418.251,Z 455.602,A -85,B 0,C 180,E1 -10045.159,E2 -10045.159} C_VEL
LIN {X 0,Y 418.237,Z 455.617,A -85,B 0,C 180,E1 -10047.472,E2 -10047.472} C_VEL
LIN {X 0,Y 418.268,Z 455.623,A -85,B 0,C 180,E1 -10050.893,E2 -10050.893} C_VEL
LIN {X 0,Y 418.262,Z 455.597,A -85,B 0,C 180,E1 -10054.096,E2 -10054.096} C_VEL
LIN {X 0,Y 418.223,Z 455.642,A -85,B 0,C 180,E1 -10057.263,E2 -10057.263} C_VEL
LIN {X 0,Y 418.274,Z 455.624,A -85,B 0,C 180,E1 -10060.364,E2 -10060.364} C_VEL
LIN {X 0,Y 418.308,Z 455.618,A -85,B 0,C 180,E1 -10063.405,E2 -10063.405} C_VEL
LIN {X 0,Y 418.337,Z 455.625,A -85,B 0,C 180,E1 -10066.999,E2 -10066.999} C_VEL
LIN {X 0,Y 418.333,Z 455.619,A -85,B 0,C 180,E1 -10070.329,E2 -10070.329} C_VEL
LIN {X 0,Y 418.485,Z 455.595,A -85,B 0,C 180,E1 -10073.249,E2 -10073.249} C_VEL
LIN {X 0,Y 418.336,Z 455.62,A -85,B 0,C 180,E1 -10075.182,E2 -10075.182} C_VEL
LIN {X 0,Y 418.536,Z 455.585,A -85,B 0,C 180,E1 -10078.076,E2 -10078.076} C_VEL
LIN {X 0,Y 418.663,Z 455.583,A -85,B 0,C 180,E1 -10080,E2 -10080} C_VEL
LIN {X 0,Y 418.503,Z 455.598,A -85,B 0,C 180,E1 -10082.888,E2 -10082.888} C_VEL
LIN {X 0,Y 418.521,Z 455.604,A -85,B 0,C 180,E1 -10085.783,E2 -10085.783} C_VEL
LIN {X 0,Y 418.392,Z 455.601,A -85,B 0,C 180,E1 -10088.695,E2 -10088.695} C_VEL
LIN {X 0,Y 418.309,Z 455.626,A -85,B 0,C 180,E1 -10091.631,E2 -10091.631} C_VEL
LIN {X 0,Y 418.294,Z 455.625,A -85,B 0,C 180,E1 -10094.597,E2 -10094.597} C_VEL
LIN {X 0,Y 418.28,Z 455.615,A -85,B 0,C 180,E1 -10097.604,E2 -10097.604} C_VEL
LIN {X 0,Y 418.241,Z 455.592,A -85,B 0,C 180,E1 -10100.663,E2 -10100.663} C_VEL
LIN {X 0,Y 418.269,Z 455.632,A -85,B 0,C 180,E1 -10103.782,E2 -10103.782} C_VEL
LIN {X 0,Y 418.303,Z 455.602,A -85,B 0,C 180,E1 -10107.071,E2 -10107.071} C_VEL
LIN {X 0,Y 418.255,Z 455.618,A -85,B 0,C 180,E1 -10110.271,E2 -10110.271} C_VEL
LIN {X 0,Y 418.243,Z 455.623,A -85,B 0,C 180,E1 -10113.678,E2 -10113.678} C_VEL
LIN {X 0,Y 418.241,Z 455.636,A -85,B 0,C 180,E1 -10117.224,E2 -10117.224} C_VEL
LIN {X 0,Y 418.259,Z 455.617,A -85,B 0,C 180,E1 -10119.681,E2 -10119.681} C_VEL
LIN {X 0,Y 418.279,Z 455.634,A -85,B 0,C 180,E1 -10122.33,E2 -10122.33} C_VEL
LIN {X 0,Y 418.248,Z 455.627,A -85,B 0,C 180,E1 -10125.112,E2 -10125.112} C_VEL
LIN {X 0,Y 418.235,Z 455.625,A -85,B 0,C 180,E1 -10127.767,E2 -10127.767} C_VEL
LIN {X 0,Y 418.258,Z 455.802,A -85,B 0,C 180,E1 -10130.242,E2 -10130.242} C_VEL
LIN {X 0,Y 421.371,Z 466.898,A -85,B 0,C 180,E1 -10132.872,E2 -10132.872} C_VEL
LIN {X 0,Y 424.844,Z 480.182,A -85,B 0,C 180,E1 -10135.724,E2 -10135.724} C_VEL
LIN {X 0,Y 428.638,Z 488.158,A -85,B 0,C 180,E1 -10136.262,E2 -10136.262} C_VEL
LIN {X 0,Y 431.439,Z 494.366,A -85,B 0,C 180,E1 -10136.629,E2 -10136.629} C_VEL
LIN {X 0,Y 438.13,Z 521.677,A -85,B 0,C 180,E1 -10137.718,E2 -10137.718} C_VEL
LIN {X 0,Y 434.513,Z 689.913,A -85,B 0,C 180,E1 -10140.608,E2 -10140.608} C_VEL
LIN {X 0,Y 433.792,Z 704.403,A -85,B 0,C 180,E1 -10140.946,E2 -10140.946} C_VEL
LIN {X 0,Y 433.019,Z 717.526,A -85,B 0,C 180,E1 -10141.377,E2 -10141.377} C_VEL
LIN {X 0,Y 432.05,Z 730.512,A -85,B 0,C 180,E1 -10141.92,E2 -10141.92} C_VEL
LIN {X 0,Y 431.068,Z 742.089,A -85,B 0,C 180,E1 -10142.51,E2 -10142.51} C_VEL
LIN {X 0,Y 429.81,Z 754.73,A -85,B 0,C 180,E1 -10143.279,E2 -10143.279} C_VEL
LIN {X 0,Y 428.564,Z 766.381,A -85,B 0,C 180,E1 -10144.113,E2 -10144.113} C_VEL
LIN {X 0,Y 427.176,Z 778.172,A -85,B 0,C 180,E1 -10145.092,E2 -10145.092} C_VEL
LIN {X 0,Y 425.805,Z 789.207,A -85,B 0,C 180,E1 -10146.148,E2 -10146.148} C_VEL
LIN {X 0,Y 424.435,Z 800.191,A -85,B 0,C 180,E1 -10147.358,E2 -10147.358} C_VEL
LIN {X 0,Y 423.179,Z 809.887,A -85,B 0,C 180,E1 -10148.57,E2 -10148.57} C_VEL
LIN {X 0,Y 421.852,Z 820.099,A -85,B 0,C 180,E1 -10150.031,E2 -10150.031} C_VEL
LIN {X 0,Y 420.734,Z 829.061,A -85,B 0,C 180,E1 -10151.496,E2 -10151.496} C_VEL
LIN {X 0,Y 419.816,Z 837.052,A -85,B 0,C 180,E1 -10152.985,E2 -10152.985} C_VEL
LIN {X 0,Y 419.066,Z 843.92,A -85,B 0,C 180,E1 -10154.435,E2 -10154.435} C_VEL
LIN {X 0,Y 418.507,Z 850.061,A -85,B 0,C 180,E1 -10155.907,E2 -10155.907} C_VEL
LIN {X 0,Y 417.896,Z 857.004,A -85,B 0,C 180,E1 -10157.865,E2 -10157.865} C_VEL
LIN {X 0,Y 417.42,Z 862.753,A -85,B 0,C 180,E1 -10159.818,E2 -10159.818} C_VEL
LIN {X 0,Y 417.258,Z 866.362,A -85,B 0,C 180,E1 -10161.281,E2 -10161.281} C_VEL
LIN {X 0,Y 417.153,Z 870.205,A -85,B 0,C 180,E1 -10163.227,E2 -10163.227} C_VEL
LIN {X 0,Y 417.042,Z 873.045,A -85,B 0,C 180,E1 -10165.167,E2 -10165.167} C_VEL
LIN {X 0,Y 417,Z 874.92,A -85,B 0,C 180,E1 -10167.102,E2 -10167.102} C_VEL
LIN {X 0,Y 417.045,Z 875.594,A -85,B 0,C 180,E1 -10168.069,E2 -10168.069} C_VEL
LIN {X 0,Y 416.959,Z 876.062,A -85,B 0,C 180,E1 -10170,E2 -10170} C_VEL
LIN {X 0,Y 417.045,Z 875.594,A -85,B 0,C 180,E1 -10171.931,E2 -10171.931} C_VEL
LIN {X 0,Y 416.97,Z 874.174,A -85,B 0,C 180,E1 -10173.866,E2 -10173.866} C_VEL
LIN {X 0,Y 417.139,Z 871.045,A -85,B 0,C 180,E1 -10176.262,E2 -10176.262} C_VEL
LIN {X 0,Y 417.215,Z 867.399,A -85,B 0,C 180,E1 -10178.232,E2 -10178.232} C_VEL
LIN {X 0,Y 417.321,Z 864.037,A -85,B 0,C 180,E1 -10179.695,E2 -10179.695} C_VEL
LIN {X 0,Y 417.714,Z 858.545,A -85,B 0,C 180,E1 -10181.648,E2 -10181.648} C_VEL
LIN {X 0,Y 418.128,Z 853.683,A -85,B 0,C 180,E1 -10183.117,E2 -10183.117} C_VEL
LIN {X 0,Y 418.861,Z 846.026,A -85,B 0,C 180,E1 -10185.074,E2 -10185.074} C_VEL
LIN {X 0,Y 419.665,Z 839.377,A -85,B 0,C 180,E1 -10186.54,E2 -10186.54} C_VEL
LIN {X 0,Y 420.438,Z 831.823,A -85,B 0,C 180,E1 -10188.013,E2 -10188.013} C_VEL
LIN {X 0,Y 421.451,Z 823.233,A -85,B 0,C 180,E1 -10189.482,E2 -10189.482} C_VEL
LIN {X 0,Y 422.749,Z 813.441,A -85,B 0,C 180,E1 -10190.942,E2 -10190.942} C_VEL
LIN {X 0,Y 424.035,Z 803.297,A -85,B 0,C 180,E1 -10192.269,E2 -10192.269} C_VEL
LIN {X 0,Y 425.316,Z 792.638,A -85,B 0,C 180,E1 -10193.493,E2 -10193.493} C_VEL
LIN {X 0,Y 426.738,Z 781.958,A -85,B 0,C 180,E1 -10194.559,E2 -10194.559} C_VEL
LIN {X 0,Y 428.022,Z 771.182,A -85,B 0,C 180,E1 -10195.505,E2 -10195.505} C_VEL
LIN {X 0,Y 429.261,Z 759.958,A -85,B 0,C 180,E1 -10196.365,E2 -10196.365} C_VEL
LIN {X 0,Y 430.545,Z 747.219,A -85,B 0,C 180,E1 -10197.197,E2 -10197.197} C_VEL
LIN {X 0,Y 431.737,Z 734.217,A -85,B 0,C 180,E1 -10197.904,E2 -10197.904} C_VEL
LIN {X 0,Y 432.809,Z 721.013,A -85,B 0,C 180,E1 -10198.488,E2 -10198.488} C_VEL
LIN {X 0,Y 433.644,Z 707.805,A -85,B 0,C 180,E1 -10198.952,E2 -10198.952} C_VEL
LIN {X 0,Y 434.339,Z 694.172,A -85,B 0,C 180,E1 -10199.305,E2 -10199.305} C_VEL
LIN {X 0,Y 435.247,Z 656.887,A -85,B 0,C 180,E1 -10199.97,E2 -10199.97} C_VEL
LIN {X 0,Y 438.072,Z 521.548,A -85,B 0,C 180,E1 -10202.289,E2 -10202.289} C_VEL
LIN {X 0,Y 431.361,Z 494.01,A -85,B 0,C 180,E1 -10203.385,E2 -10203.385} C_VEL
LIN {X 0,Y 424.913,Z 480.385,A -85,B 0,C 180,E1 -10204.25,E2 -10204.25} C_VEL
LIN {X 0,Y 422.082,Z 469.506,A -85,B 0,C 180,E1 -10206.544,E2 -10206.544} C_VEL
LIN {X 0,Y 418.31,Z 456.029,A -85,B 0,C 180,E1 -10209.674,E2 -10209.674} C_VEL
LIN {X 0,Y 418.243,Z 455.617,A -85,B 0,C 180,E1 -10209.995,E2 -10209.995} C_VEL
LIN {X 0,Y 418.224,Z 455.627,A -85,B 0,C 180,E1 -10212.32,E2 -10212.32} C_VEL
LIN {X 0,Y 418.255,Z 455.624,A -85,B 0,C 180,E1 -10215.111,E2 -10215.111} C_VEL
LIN {X 0,Y 418.286,Z 455.635,A -85,B 0,C 180,E1 -10217.773,E2 -10217.773} C_VEL
LIN {X 0,Y 418.26,Z 455.629,A -85,B 0,C 180,E1 -10221.559,E2 -10221.559} C_VEL
LIN {X 0,Y 418.253,Z 455.609,A -85,B 0,C 180,E1 -10225.158,E2 -10225.158} C_VEL
LIN {X 0,Y 418.242,Z 455.634,A -85,B 0,C 180,E1 -10227.472,E2 -10227.472} C_VEL
LIN {X 0,Y 418.269,Z 455.598,A -85,B 0,C 180,E1 -10230.893,E2 -10230.893} C_VEL
LIN {X 0,Y 418.264,Z 455.623,A -85,B 0,C 180,E1 -10234.095,E2 -10234.095} C_VEL
LIN {X 0,Y 418.224,Z 455.631,A -85,B 0,C 180,E1 -10237.263,E2 -10237.263} C_VEL
LIN {X 0,Y 418.275,Z 455.587,A -85,B 0,C 180,E1 -10240.364,E2 -10240.364} C_VEL
LIN {X 0,Y 418.309,Z 455.622,A -85,B 0,C 180,E1 -10243.404,E2 -10243.404} C_VEL
LIN {X 0,Y 418.338,Z 455.613,A -85,B 0,C 180,E1 -10246.999,E2 -10246.999} C_VEL
LIN {X 0,Y 418.334,Z 455.618,A -85,B 0,C 180,E1 -10250.328,E2 -10250.328} C_VEL
LIN {X 0,Y 418.484,Z 455.604,A -85,B 0,C 180,E1 -10253.249,E2 -10253.249} C_VEL
LIN {X 0,Y 418.334,Z 455.618,A -85,B 0,C 180,E1 -10255.181,E2 -10255.181} C_VEL
LIN {X 0,Y 418.536,Z 455.596,A -85,B 0,C 180,E1 -10258.075,E2 -10258.075} C_VEL
LIN {X 0,Y 418.663,Z 455.583,A -85,B 0,C 180,E1 -10260,E2 -10260} C_VEL
LIN {X 0,Y 418.503,Z 455.601,A -85,B 0,C 180,E1 -10262.888,E2 -10262.888} C_VEL
LIN {X 0,Y 418.485,Z 455.594,A -85,B 0,C 180,E1 -10266.751,E2 -10266.751} C_VEL
LIN {X 0,Y 418.333,Z 455.618,A -85,B 0,C 180,E1 -10269.671,E2 -10269.671} C_VEL
LIN {X 0,Y 418.337,Z 455.625,A -85,B 0,C 180,E1 -10273.001,E2 -10273.001} C_VEL
LIN {X 0,Y 418.304,Z 455.62,A -85,B 0,C 180,E1 -10276.735,E2 -10276.735} C_VEL
LIN {X 0,Y 418.262,Z 455.626,A -85,B 0,C 180,E1 -10279.79,E2 -10279.79} C_VEL
LIN {X 0,Y 418.223,Z 455.642,A -85,B 0,C 180,E1 -10282.737,E2 -10282.737} C_VEL
LIN {X 0,Y 418.262,Z 455.597,A -85,B 0,C 180,E1 -10285.904,E2 -10285.904} C_VEL
LIN {X 0,Y 418.266,Z 455.625,A -85,B 0,C 180,E1 -10289.161,E2 -10289.161} C_VEL
LIN {X 0,Y 418.249,Z 455.609,A -85,B 0,C 180,E1 -10292.844,E2 -10292.844} C_VEL
LIN {X 0,Y 418.241,Z 455.631,A -85,B 0,C 180,E1 -10296.239,E2 -10296.239} C_VEL
LIN {X 0,Y 418.259,Z 455.636,A -85,B 0,C 180,E1 -10299.68,E2 -10299.68} C_VEL
LIN {X 0,Y 418.278,Z 455.632,A -85,B 0,C 180,E1 -10302.33,E2 -10302.33} C_VEL
LIN {X 0,Y 418.244,Z 455.639,A -85,B 0,C 180,E1 -10305.111,E2 -10305.111} C_VEL
LIN {X 0,Y 418.249,Z 455.637,A -85,B 0,C 180,E1 -10307.769,E2 -10307.769} C_VEL
LIN {X 0,Y 418.261,Z 455.634,A -85,B 0,C 180,E1 -10310.617,E2 -10310.617} C_VEL
LIN {X 0,Y 418.24,Z 455.636,A -85,B 0,C 180,E1 -10313.977,E2 -10313.977} C_VEL
LIN {X 0,Y 418.252,Z 455.637,A -85,B 0,C 180,E1 -10317.156,E2 -10317.156} C_VEL
LIN {X 0,Y 418.263,Z 455.636,A -85,B 0,C 180,E1 -10320.896,E2 -10320.896} C_VEL
LIN {X 0,Y 418.266,Z 455.633,A -85,B 0,C 180,E1 -10324.096,E2 -10324.096} C_VEL
LIN {X 0,Y 418.234,Z 455.638,A -85,B 0,C 180,E1 -10327.264,E2 -10327.264} C_VEL
LIN {X 0,Y 418.279,Z 455.634,A -85,B 0,C 180,E1 -10330.364,E2 -10330.364} C_VEL
LIN {X 0,Y 418.313,Z 455.63,A -85,B 0,C 180,E1 -10333.405,E2 -10333.405} C_VEL
LIN {X 0,Y 418.352,Z 455.623,A -85,B 0,C 180,E1 -10336.994,E2 -10336.994} C_VEL
LIN {X 0,Y 418.356,Z 455.625,A -85,B 0,C 180,E1 -10340.329,E2 -10340.329} C_VEL
LIN {X 0,Y 418.49,Z 455.609,A -85,B 0,C 180,E1 -10343.249,E2 -10343.249} C_VEL
LIN {X 0,Y 418.337,Z 455.625,A -85,B 0,C 180,E1 -10345.182,E2 -10345.182} C_VEL
LIN {X 0,Y 418.541,Z 455.6,A -85,B 0,C 180,E1 -10348.076,E2 -10348.076} C_VEL
LIN {X 0,Y 418.669,Z 455.587,A -85,B 0,C 180,E1 -10350,E2 -10350} C_VEL
LIN {X 0,Y 418.508,Z 455.606,A -85,B 0,C 180,E1 -10352.888,E2 -10352.888} C_VEL
LIN {X 0,Y 418.49,Z 455.608,A -85,B 0,C 180,E1 -10356.751,E2 -10356.751} C_VEL
LIN {X 0,Y 418.356,Z 455.625,A -85,B 0,C 180,E1 -10359.671,E2 -10359.671} C_VEL
LIN {X 0,Y 418.352,Z 455.623,A -85,B 0,C 180,E1 -10363.006,E2 -10363.006} C_VEL
LIN {X 0,Y 418.329,Z 455.626,A -85,B 0,C 180,E1 -10363.344,E2 -10363.344} C_VEL
LIN {X 0,Y 417.637,Z 455.715,A -85,B 0,C 180,E1 -10364.147,E2 -10364.147} C_VEL
LIN {X 0,Y 414.754,Z 456.072,A -85,B 0,C 180,E1 -10365.452,E2 -10365.452} C_VEL
LIN {X 0,Y 412.336,Z 456.376,A -85,B 0,C 180,E1 -10366.506,E2 -10366.506} C_VEL
LIN {X 0,Y 411.312,Z 456.499,A -85,B 0,C 180,E1 -10367.321,E2 -10367.321} C_VEL
LIN {X 0,Y 411.236,Z 456.509,A -85,B 0,C 180,E1 -10367.597,E2 -10367.597} C_VEL
LIN {X 0,Y 411.192,Z 456.515,A -85,B 0,C 180,E1 -10371.034,E2 -10371.034} C_VEL
LIN {X 0,Y 411.222,Z 456.512,A -85,B 0,C 180,E1 -10374.215,E2 -10374.215} C_VEL
LIN {X 0,Y 411.254,Z 456.508,A -85,B 0,C 180,E1 -10377.477,E2 -10377.477} C_VEL
LIN {X 0,Y 411.184,Z 456.517,A -85,B 0,C 180,E1 -10380.847,E2 -10380.847} C_VEL
LIN {X 0,Y 411.2,Z 456.514,A -85,B 0,C 180,E1 -10384.333,E2 -10384.333} C_VEL
LIN {X 0,Y 411.198,Z 456.516,A -85,B 0,C 180,E1 -10387.972,E2 -10387.972} C_VEL
LIN {X 0,Y 411.193,Z 456.514,A -85,B 0,C 180,E1 -10391.234,E2 -10391.234} C_VEL
LIN {X 0,Y 411.177,Z 456.518,A -85,B 0,C 180,E1 -10394.489,E2 -10394.489} C_VEL
LIN {X 0,Y 411.226,Z 456.512,A -85,B 0,C 180,E1 -10397.296,E2 -10397.296} C_VEL
LIN {X 0,Y 411.224,Z 456.514,A -85,B 0,C 180,E1 -10400.777,E2 -10400.777} C_VEL
LIN {X 0,Y 411.192,Z 456.492,A -85,B 0,C 180,E1 -10404.471,E2 -10404.471} C_VEL
LIN {X 0,Y 411.199,Z 456.481,A -85,B 0,C 180,E1 -10406.873,E2 -10406.873} C_VEL
LIN {X 0,Y 411.233,Z 456.504,A -85,B 0,C 180,E1 -10410.642,E2 -10410.642} C_VEL
LIN {X 0,Y 411.229,Z 456.468,A -85,B 0,C 180,E1 -10413.619,E2 -10413.619} C_VEL
LIN {X 0,Y 411.188,Z 456.513,A -85,B 0,C 180,E1 -10416.852,E2 -10416.852} C_VEL
LIN {X 0,Y 411.206,Z 456.504,A -85,B 0,C 180,E1 -10420.05,E2 -10420.05} C_VEL
LIN {X 0,Y 411.254,Z 456.5,A -85,B 0,C 180,E1 -10423.131,E2 -10423.131} C_VEL
LIN {X 0,Y 411.296,Z 456.501,A -85,B 0,C 180,E1 -10426.896,E2 -10426.896} C_VEL
LIN {X 0,Y 411.285,Z 456.498,A -85,B 0,C 180,E1 -10430.161,E2 -10430.161} C_VEL
LIN {X 0,Y 411.448,Z 456.472,A -85,B 0,C 180,E1 -10433.133,E2 -10433.133} C_VEL
LIN {X 0,Y 411.306,Z 456.494,A -85,B 0,C 180,E1 -10435.099,E2 -10435.099} C_VEL
LIN {X 0,Y 411.505,Z 456.461,A -85,B 0,C 180,E1 -10438.043,E2 -10438.043} C_VEL
LIN {X 0,Y 411.633,Z 456.459,A -85,B 0,C 180,E1 -10440,E2 -10440} C_VEL
LIN {X 0,Y 411.458,Z 456.474,A -85,B 0,C 180,E1 -10442.937,E2 -10442.937} C_VEL
LIN {X 0,Y 411.48,Z 456.48,A -85,B 0,C 180,E1 -10445.882,E2 -10445.882} C_VEL
LIN {X 0,Y 411.346,Z 456.479,A -85,B 0,C 180,E1 -10448.846,E2 -10448.846} C_VEL
LIN {X 0,Y 411.277,Z 456.499,A -85,B 0,C 180,E1 -10451.833,E2 -10451.833} C_VEL
LIN {X 0,Y 411.251,Z 456.502,A -85,B 0,C 180,E1 -10454.853,E2 -10454.853} C_VEL
LIN {X 0,Y 411.244,Z 456.486,A -85,B 0,C 180,E1 -10457.916,E2 -10457.916} C_VEL
LIN {X 0,Y 411.188,Z 456.473,A -85,B 0,C 180,E1 -10461.035,E2 -10461.035} C_VEL
LIN {X 0,Y 411.214,Z 456.514,A -85,B 0,C 180,E1 -10464.216,E2 -10464.216} C_VEL
LIN {X 0,Y 411.253,Z 456.472,A -85,B 0,C 180,E1 -10467.478,E2 -10467.478} C_VEL
LIN {X 0,Y 411.193,Z 456.511,A -85,B 0,C 180,E1 -10470.847,E2 -10470.847} C_VEL
LIN {X 0,Y 411.2,Z 456.49,A -85,B 0,C 180,E1 -10474.334,E2 -10474.334} C_VEL
LIN {X 0,Y 411.199,Z 456.516,A -85,B 0,C 180,E1 -10477.973,E2 -10477.973} C_VEL
LIN {X 0,Y 411.204,Z 456.506,A -85,B 0,C 180,E1 -10481.236,E2 -10481.236} C_VEL
LIN {X 0,Y 411.219,Z 456.496,A -85,B 0,C 180,E1 -10484.484,E2 -10484.484} C_VEL
LIN {X 0,Y 411.172,Z 456.506,A -85,B 0,C 180,E1 -10488.195,E2 -10488.195} C_VEL
LIN {X 0,Y 411.226,Z 456.568,A -85,B 0,C 180,E1 -10489.609,E2 -10489.609} C_VEL
LIN {X 0,Y 411.755,Z 458.612,A -85,B 0,C 180,E1 -10490.181,E2 -10490.181} C_VEL
LIN {X 0,Y 415.241,Z 471.111,A -85,B 0,C 180,E1 -10493.133,E2 -10493.133} C_VEL
LIN {X 0,Y 417.607,Z 480.04,A -85,B 0,C 180,E1 -10495.061,E2 -10495.061} C_VEL
LIN {X 0,Y 425.664,Z 496.655,A -85,B 0,C 180,E1 -10496.165,E2 -10496.165} C_VEL
LIN {X 0,Y 432.055,Z 522.928,A -85,B 0,C 180,E1 -10497.236,E2 -10497.236} C_VEL
LIN {X 0,Y 428.79,Z 671.006,A -85,B 0,C 180,E1 -10499.804,E2 -10499.804} C_VEL
LIN {X 0,Y 428.045,Z 696.802,A -85,B 0,C 180,E1 -10500.289,E2 -10500.289} C_VEL
LIN {X 0,Y 426.93,Z 715.054,A -85,B 0,C 180,E1 -10500.83,E2 -10500.83} C_VEL
LIN {X 0,Y 425.901,Z 729.068,A -85,B 0,C 180,E1 -10501.41,E2 -10501.41} C_VEL
LIN {X 0,Y 424.713,Z 741.877,A -85,B 0,C 180,E1 -10502.063,E2 -10502.063} C_VEL
LIN {X 0,Y 423.44,Z 754.519,A -85,B 0,C 180,E1 -10502.844,E2 -10502.844} C_VEL
LIN {X 0,Y 422.141,Z 766.165,A -85,B 0,C 180,E1 -10503.688,E2 -10503.688} C_VEL
LIN {X 0,Y 420.702,Z 777.816,A -85,B 0,C 180,E1 -10504.668,E2 -10504.668} C_VEL
LIN {X 0,Y 419.232,Z 788.994,A -85,B 0,C 180,E1 -10505.751,E2 -10505.751} C_VEL
LIN {X 0,Y 417.805,Z 799.979,A -85,B 0,C 180,E1 -10506.978,E2 -10506.978} C_VEL
LIN {X 0,Y 416.478,Z 809.674,A -85,B 0,C 180,E1 -10508.208,E2 -10508.208} C_VEL
LIN {X 0,Y 415.073,Z 819.886,A -85,B 0,C 180,E1 -10509.69,E2 -10509.69} C_VEL
LIN {X 0,Y 413.893,Z 828.847,A -85,B 0,C 180,E1 -10511.179,E2 -10511.179} C_VEL
LIN {X 0,Y 412.878,Z 837.006,A -85,B 0,C 180,E1 -10512.726,E2 -10512.726} C_VEL
LIN {X 0,Y 412.133,Z 843.707,A -85,B 0,C 180,E1 -10514.167,E2 -10514.167} C_VEL
LIN {X 0,Y 411.515,Z 849.848,A -85,B 0,C 180,E1 -10515.663,E2 -10515.663} C_VEL
LIN {X 0,Y 410.879,Z 856.792,A -85,B 0,C 180,E1 -10517.655,E2 -10517.655} C_VEL
LIN {X 0,Y 410.356,Z 862.541,A -85,B 0,C 180,E1 -10519.64,E2 -10519.64} C_VEL
LIN {X 0,Y 410.19,Z 866.15,A -85,B 0,C 180,E1 -10521.13,E2 -10521.13} C_VEL
LIN {X 0,Y 410.057,Z 869.994,A -85,B 0,C 180,E1 -10523.11,E2 -10523.11} C_VEL
LIN {X 0,Y 409.953,Z 872.834,A -85,B 0,C 180,E1 -10525.083,E2 -10525.083} C_VEL
LIN {X 0,Y 409.898,Z 874.71,A -85,B 0,C 180,E1 -10527.052,E2 -10527.052} C_VEL
LIN {X 0,Y 409.955,Z 875.384,A -85,B 0,C 180,E1 -10528.035,E2 -10528.035} C_VEL
LIN {X 0,Y 409.884,Z 875.853,A -85,B 0,C 180,E1 -10530,E2 -10530} C_VEL
LIN {X 0,Y 409.955,Z 875.384,A -85,B 0,C 180,E1 -10531.965,E2 -10531.965} C_VEL
LIN {X 0,Y 409.888,Z 873.964,A -85,B 0,C 180,E1 -10533.933,E2 -10533.933} C_VEL
LIN {X 0,Y 410.04,Z 871.07,A -85,B 0,C 180,E1 -10536.225,E2 -10536.225} C_VEL
LIN {X 0,Y 410.129,Z 867.188,A -85,B 0,C 180,E1 -10538.375,E2 -10538.375} C_VEL
LIN {X 0,Y 410.251,Z 863.825,A -85,B 0,C 180,E1 -10539.864,E2 -10539.864} C_VEL
LIN {X 0,Y 410.681,Z 858.333,A -85,B 0,C 180,E1 -10541.85,E2 -10541.85} C_VEL
LIN {X 0,Y 411.109,Z 853.66,A -85,B 0,C 180,E1 -10543.293,E2 -10543.293} C_VEL
LIN {X 0,Y 411.892,Z 845.813,A -85,B 0,C 180,E1 -10545.335,E2 -10545.335} C_VEL
LIN {X 0,Y 412.752,Z 839.164,A -85,B 0,C 180,E1 -10546.825,E2 -10546.825} C_VEL
LIN {X 0,Y 413.571,Z 831.607,A -85,B 0,C 180,E1 -10548.323,E2 -10548.323} C_VEL
LIN {X 0,Y 414.659,Z 823.019,A -85,B 0,C 180,E1 -10549.814,E2 -10549.814} C_VEL
LIN {X 0,Y 416.019,Z 813.227,A -85,B 0,C 180,E1 -10551.297,E2 -10551.297} C_VEL
LIN {X 0,Y 417.356,Z 803,A -85,B 0,C 180,E1 -10552.655,E2 -10552.655} C_VEL
LIN {X 0,Y 418.741,Z 792.426,A -85,B 0,C 180,E1 -10553.885,E2 -10553.885} C_VEL
LIN {X 0,Y 420.169,Z 781.952,A -85,B 0,C 180,E1 -10554.948,E2 -10554.948} C_VEL
LIN {X 0,Y 421.527,Z 770.969,A -85,B 0,C 180,E1 -10555.927,E2 -10555.927} C_VEL
LIN {X 0,Y 422.852,Z 759.746,A -85,B 0,C 180,E1 -10556.796,E2 -10556.796} C_VEL
LIN {X 0,Y 424.206,Z 747.008,A -85,B 0,C 180,E1 -10557.638,E2 -10557.638} C_VEL
LIN {X 0,Y 425.432,Z 734.006,A -85,B 0,C 180,E1 -10558.355,E2 -10558.355} C_VEL
LIN {X 0,Y 426.608,Z 720.12,A -85,B 0,C 180,E1 -10558.971,E2 -10558.971} C_VEL
LIN {X 0,Y 427.453,Z 707.075,A -85,B 0,C 180,E1 -10559.43,E2 -10559.43} C_VEL
LIN {X 0,Y 428.165,Z 693.963,A -85,B 0,C 180,E1 -10559.77,E2 -10559.77} C_VEL
LIN {X 0,Y 429.101,Z 656.677,A -85,B 0,C 180,E1 -10560.444,E2 -10560.444} C_VEL
LIN {X 0,Y 432.091,Z 524.125,A -85,B 0,C 180,E1 -10562.738,E2 -10562.738} C_VEL
LIN {X 0,Y 431.42,Z 520.543,A -85,B 0,C 180,E1 -10562.864,E2 -10562.864} C_VEL
LIN {X 0,Y 425.799,Z 497.112,A -85,B 0,C 180,E1 -10563.814,E2 -10563.814} C_VEL
LIN {X 0,Y 417.57,Z 479.992,A -85,B 0,C 180,E1 -10564.947,E2 -10564.947} C_VEL
LIN {X 0,Y 414.808,Z 469.567,A -85,B 0,C 180,E1 -10567.221,E2 -10567.221} C_VEL
LIN {X 0,Y 411.334,Z 457.148,A -85,B 0,C 180,E1 -10570.179,E2 -10570.179} C_VEL
LIN {X 0,Y 411.198,Z 456.522,A -85,B 0,C 180,E1 -10570.501,E2 -10570.501} C_VEL
LIN {X 0,Y 411.169,Z 456.52,A -85,B 0,C 180,E1 -10574.119,E2 -10574.119} C_VEL
LIN {X 0,Y 411.223,Z 456.509,A -85,B 0,C 180,E1 -10577.296,E2 -10577.296} C_VEL
LIN {X 0,Y 411.225,Z 456.497,A -85,B 0,C 180,E1 -10580.777,E2 -10580.777} C_VEL
LIN {X 0,Y 411.193,Z 456.49,A -85,B 0,C 180,E1 -10584.471,E2 -10584.471} C_VEL
LIN {X 0,Y 411.165,Z 456.521,A -85,B 0,C 180,E1 -10588.003,E2 -10588.003} C_VEL
LIN {X 0,Y 411.216,Z 456.471,A -85,B 0,C 180,E1 -10591.41,E2 -10591.41} C_VEL
LIN {X 0,Y 411.231,Z 456.492,A -85,B 0,C 180,E1 -10593.619,E2 -10593.619} C_VEL
LIN {X 0,Y 411.189,Z 456.508,A -85,B 0,C 180,E1 -10596.852,E2 -10596.852} C_VEL
LIN {X 0,Y 411.206,Z 456.464,A -85,B 0,C 180,E1 -10600.05,E2 -10600.05} C_VEL
LIN {X 0,Y 411.255,Z 456.5,A -85,B 0,C 180,E1 -10603.131,E2 -10603.131} C_VEL
LIN {X 0,Y 411.297,Z 456.489,A -85,B 0,C 180,E1 -10606.896,E2 -10606.896} C_VEL
LIN {X 0,Y 411.286,Z 456.498,A -85,B 0,C 180,E1 -10610.161,E2 -10610.161} C_VEL
LIN {X 0,Y 411.447,Z 456.481,A -85,B 0,C 180,E1 -10613.133,E2 -10613.133} C_VEL
LIN {X 0,Y 411.306,Z 456.494,A -85,B 0,C 180,E1 -10615.099,E2 -10615.099} C_VEL
LIN {X 0,Y 411.505,Z 456.471,A -85,B 0,C 180,E1 -10618.042,E2 -10618.042} C_VEL
LIN {X 0,Y 411.633,Z 456.458,A -85,B 0,C 180,E1 -10620,E2 -10620} C_VEL
LIN {X 0,Y 411.459,Z 456.479,A -85,B 0,C 180,E1 -10622.937,E2 -10622.937} C_VEL
LIN {X 0,Y 411.448,Z 456.47,A -85,B 0,C 180,E1 -10626.867,E2 -10626.867} C_VEL
LIN {X 0,Y 411.285,Z 456.497,A -85,B 0,C 180,E1 -10629.839,E2 -10629.839} C_VEL
LIN {X 0,Y 411.296,Z 456.501,A -85,B 0,C 180,E1 -10633.104,E2 -10633.104} C_VEL
LIN {X 0,Y 411.254,Z 456.5,A -85,B 0,C 180,E1 -10636.869,E2 -10636.869} C_VEL
LIN {X 0,Y 411.222,Z 456.502,A -85,B 0,C 180,E1 -10639.987,E2 -10639.987} C_VEL
LIN {X 0,Y 411.188,Z 456.513,A -85,B 0,C 180,E1 -10643.148,E2 -10643.148} C_VEL
LIN {X 0,Y 411.229,Z 456.468,A -85,B 0,C 180,E1 -10646.381,E2 -10646.381} C_VEL
LIN {X 0,Y 411.203,Z 456.513,A -85,B 0,C 180,E1 -10649.712,E2 -10649.712} C_VEL
LIN {X 0,Y 411.198,Z 456.48,A -85,B 0,C 180,E1 -10653.156,E2 -10653.156} C_VEL
LIN {X 0,Y 411.188,Z 456.511,A -85,B 0,C 180,E1 -10656.553,E2 -10656.553} C_VEL
LIN {X 0,Y 411.221,Z 456.512,A -85,B 0,C 180,E1 -10659.731,E2 -10659.731} C_VEL
LIN {X 0,Y 411.224,Z 456.514,A -85,B 0,C 180,E1 -10663.126,E2 -10663.126} C_VEL
LIN {X 0,Y 411.165,Z 456.52,A -85,B 0,C 180,E1 -10665.881,E2 -10665.881} C_VEL
LIN {X 0,Y 411.205,Z 456.515,A -85,B 0,C 180,E1 -10669.5,E2 -10669.5} C_VEL
LIN {X 0,Y 411.198,Z 456.516,A -85,B 0,C 180,E1 -10672.028,E2 -10672.028} C_VEL
LIN {X 0,Y 411.2,Z 456.514,A -85,B 0,C 180,E1 -10675.667,E2 -10675.667} C_VEL
LIN {X 0,Y 411.184,Z 456.517,A -85,B 0,C 180,E1 -10679.153,E2 -10679.153} C_VEL
LIN {X 0,Y 411.254,Z 456.508,A -85,B 0,C 180,E1 -10682.523,E2 -10682.523} C_VEL
LIN {X 0,Y 411.222,Z 456.511,A -85,B 0,C 180,E1 -10685.785,E2 -10685.785} C_VEL
LIN {X 0,Y 411.192,Z 456.515,A -85,B 0,C 180,E1 -10688.966,E2 -10688.966} C_VEL
LIN {X 0,Y 411.249,Z 456.51,A -85,B 0,C 180,E1 -10692.085,E2 -10692.085} C_VEL
LIN {X 0,Y 411.258,Z 456.508,A -85,B 0,C 180,E1 -10695.148,E2 -10695.148} C_VEL
LIN {X 0,Y 411.295,Z 456.502,A -85,B 0,C 180,E1 -10698.168,E2 -10698.168} C_VEL
LIN {X 0,Y 411.479,Z 456.48,A -85,B 0,C 180,E1 -10702.147,E2 -10702.147} C_VEL
LIN {X 0,Y 411.472,Z 456.481,A -85,B 0,C 180,E1 -10704.118,E2 -10704.118} C_VEL
LIN {X 0,Y 411.511,Z 456.476,A -85,B 0,C 180,E1 -10708.043,E2 -10708.043} C_VEL
LIN {X 0,Y 411.639,Z 456.463,A -85,B 0,C 180,E1 -10710,E2 -10710} C_VEL
LIN {X 0,Y 411.463,Z 456.483,A -85,B 0,C 180,E1 -10712.937,E2 -10712.937} C_VEL
LIN {X 0,Y 411.457,Z 456.484,A -85,B 0,C 180,E1 -10716.867,E2 -10716.867} C_VEL
LIN {X 0,Y 411.304,Z 456.503,A -85,B 0,C 180,E1 -10719.838,E2 -10719.838} C_VEL
LIN {X 0,Y 411.288,Z 456.503,A -85,B 0,C 180,E1 -10723.332,E2 -10723.332} C_VEL
LIN {X 0,Y 411.253,Z 456.507,A -85,B 0,C 180,E1 -10726.888,E2 -10726.888} C_VEL
LIN {X 0,Y 411.236,Z 456.509,A -85,B 0,C 180,E1 -10727.597,E2 -10727.597} C_VEL
LIN {X 0,Y 410.576,Z 456.594,A -85,B 0,C 180,E1 -10728.415,E2 -10728.415} C_VEL
LIN {X 0,Y 407.688,Z 456.953,A -85,B 0,C 180,E1 -10729.743,E2 -10729.743} C_VEL
LIN {X 0,Y 405.243,Z 457.258,A -85,B 0,C 180,E1 -10730.816,E2 -10730.816} C_VEL
LIN {X 0,Y 404.208,Z 457.385,A -85,B 0,C 180,E1 -10731.646,E2 -10731.646} C_VEL
LIN {X 0,Y 404.131,Z 457.392,A -85,B 0,C 180,E1 -10731.927,E2 -10731.927} C_VEL
LIN {X 0,Y 404.211,Z 457.385,A -85,B 0,C 180,E1 -10735.296,E2 -10735.296} C_VEL
LIN {X 0,Y 404.19,Z 457.389,A -85,B 0,C 180,E1 -10737.999,E2 -10737.999} C_VEL
LIN {X 0,Y 404.134,Z 457.394,A -85,B 0,C 180,E1 -10741.558,E2 -10741.558} C_VEL
LIN {X 0,Y 404.18,Z 457.389,A -85,B 0,C 180,E1 -10745.016,E2 -10745.016} C_VEL
LIN {X 0,Y 404.157,Z 457.393,A -85,B 0,C 180,E1 -10748.756,E2 -10748.756} C_VEL
LIN {X 0,Y 404.143,Z 457.393,A -85,B 0,C 180,E1 -10751.604,E2 -10751.604} C_VEL
LIN {X 0,Y 404.146,Z 457.393,A -85,B 0,C 180,E1 -10754.523,E2 -10754.523} C_VEL
LIN {X 0,Y 404.204,Z 457.387,A -85,B 0,C 180,E1 -10757.305,E2 -10757.305} C_VEL
LIN {X 0,Y 404.161,Z 457.391,A -85,B 0,C 180,E1 -10759.955,E2 -10759.955} C_VEL
LIN {X 0,Y 404.133,Z 457.393,A -85,B 0,C 180,E1 -10763.124,E2 -10763.124} C_VEL
LIN {X 0,Y 404.137,Z 457.353,A -85,B 0,C 180,E1 -10766.187,E2 -10766.187} C_VEL
LIN {X 0,Y 404.146,Z 457.392,A -85,B 0,C 180,E1 -10769.715,E2 -10769.715} C_VEL
LIN {X 0,Y 404.187,Z 457.343,A -85,B 0,C 180,E1 -10773.123,E2 -10773.123} C_VEL
LIN {X 0,Y 404.166,Z 457.369,A -85,B 0,C 180,E1 -10775.334,E2 -10775.334} C_VEL
LIN {X 0,Y 404.129,Z 457.392,A -85,B 0,C 180,E1 -10778.581,E2 -10778.581} C_VEL
LIN {X 0,Y 404.201,Z 457.385,A -85,B 0,C 180,E1 -10781.762,E2 -10781.762} C_VEL
LIN {X 0,Y 404.197,Z 457.374,A -85,B 0,C 180,E1 -10784.882,E2 -10784.882} C_VEL
LIN {X 0,Y 404.248,Z 457.368,A -85,B 0,C 180,E1 -10787.959,E2 -10787.959} C_VEL
LIN {X 0,Y 404.396,Z 457.354,A -85,B 0,C 180,E1 -10792.129,E2 -10792.129} C_VEL
LIN {X 0,Y 404.416,Z 457.346,A -85,B 0,C 180,E1 -10794.015,E2 -10794.015} C_VEL
LIN {X 0,Y 404.474,Z 457.337,A -85,B 0,C 180,E1 -10798.009,E2 -10798.009} C_VEL
LIN {X 0,Y 404.602,Z 457.334,A -85,B 0,C 180,E1 -10800,E2 -10800} C_VEL
LIN {X 0,Y 404.415,Z 457.35,A -85,B 0,C 180,E1 -10802.989,E2 -10802.989} C_VEL
LIN {X 0,Y 404.426,Z 457.357,A -85,B 0,C 180,E1 -10805.985,E2 -10805.985} C_VEL
LIN {X 0,Y 404.283,Z 457.359,A -85,B 0,C 180,E1 -10809.001,E2 -10809.001} C_VEL
LIN {X 0,Y 404.249,Z 457.371,A -85,B 0,C 180,E1 -10812.042,E2 -10812.042} C_VEL
LIN {X 0,Y 404.198,Z 457.382,A -85,B 0,C 180,E1 -10815.118,E2 -10815.118} C_VEL
LIN {X 0,Y 404.202,Z 457.358,A -85,B 0,C 180,E1 -10818.239,E2 -10818.239} C_VEL
LIN {X 0,Y 404.13,Z 457.357,A -85,B 0,C 180,E1 -10821.42,E2 -10821.42} C_VEL
LIN {X 0,Y 404.167,Z 457.388,A -85,B 0,C 180,E1 -10824.666,E2 -10824.666} C_VEL
LIN {X 0,Y 404.191,Z 457.345,A -85,B 0,C 180,E1 -10828,E2 -10828} C_VEL
LIN {X 0,Y 404.139,Z 457.392,A -85,B 0,C 180,E1 -10831.56,E2 -10831.56} C_VEL
LIN {X 0,Y 404.179,Z 457.361,A -85,B 0,C 180,E1 -10835.017,E2 -10835.017} C_VEL
LIN {X 0,Y 404.158,Z 457.383,A -85,B 0,C 180,E1 -10838.757,E2 -10838.757} C_VEL
LIN {X 0,Y 404.185,Z 457.385,A -85,B 0,C 180,E1 -10841.611,E2 -10841.611} C_VEL
LIN {X 0,Y 404.185,Z 457.372,A -85,B 0,C 180,E1 -10844.529,E2 -10844.529} C_VEL
LIN {X 0,Y 404.132,Z 457.382,A -85,B 0,C 180,E1 -10847.296,E2 -10847.296} C_VEL
LIN {X 0,Y 404.144,Z 457.559,A -85,B 0,C 180,E1 -10849.062,E2 -10849.062} C_VEL
LIN {X 0,Y 407,Z 467.505,A -85,B 0,C 180,E1 -10851.565,E2 -10851.565} C_VEL
LIN {X 0,Y 410.263,Z 479.645,A -85,B 0,C 180,E1 -10854.333,E2 -10854.333} C_VEL
LIN {X 0,Y 419.412,Z 498.336,A -85,B 0,C 180,E1 -10855.629,E2 -10855.629} C_VEL
LIN {X 0,Y 420.454,Z 501.012,A -85,B 0,C 180,E1 -10855.779,E2 -10855.779} C_VEL
LIN {X 0,Y 426.034,Z 524.424,A -85,B 0,C 180,E1 -10856.747,E2 -10856.747} C_VEL
LIN {X 0,Y 422.897,Z 660.049,A -85,B 0,C 180,E1 -10859.13,E2 -10859.13} C_VEL
LIN {X 0,Y 421.993,Z 693.752,A -85,B 0,C 180,E1 -10859.75,E2 -10859.75} C_VEL
LIN {X 0,Y 421.186,Z 708.289,A -85,B 0,C 180,E1 -10860.137,E2 -10860.137} C_VEL
LIN {X 0,Y 419.972,Z 724.892,A -85,B 0,C 180,E1 -10860.751,E2 -10860.751} C_VEL
LIN {X 0,Y 418.421,Z 741.666,A -85,B 0,C 180,E1 -10861.606,E2 -10861.606} C_VEL
LIN {X 0,Y 417.096,Z 754.308,A -85,B 0,C 180,E1 -10862.396,E2 -10862.396} C_VEL
LIN {X 0,Y 415.73,Z 765.953,A -85,B 0,C 180,E1 -10863.251,E2 -10863.251} C_VEL
LIN {X 0,Y 414.135,Z 778.26,A -85,B 0,C 180,E1 -10864.305,E2 -10864.305} C_VEL
LIN {X 0,Y 412.522,Z 789.926,A -85,B 0,C 180,E1 -10865.464,E2 -10865.464} C_VEL
LIN {X 0,Y 411.167,Z 799.765,A -85,B 0,C 180,E1 -10866.584,E2 -10866.584} C_VEL
LIN {X 0,Y 409.584,Z 810.821,A -85,B 0,C 180,E1 -10868.025,E2 -10868.025} C_VEL
LIN {X 0,Y 408.304,Z 819.672,A -85,B 0,C 180,E1 -10869.338,E2 -10869.338} C_VEL
LIN {X 0,Y 407.054,Z 828.634,A -85,B 0,C 180,E1 -10870.85,E2 -10870.85} C_VEL
LIN {X 0,Y 405.954,Z 837.074,A -85,B 0,C 180,E1 -10872.482,E2 -10872.482} C_VEL
LIN {X 0,Y 405.205,Z 843.494,A -85,B 0,C 180,E1 -10873.889,E2 -10873.889} C_VEL
LIN {X 0,Y 404.529,Z 849.635,A -85,B 0,C 180,E1 -10875.41,E2 -10875.41} C_VEL
LIN {X 0,Y 403.843,Z 856.618,A -85,B 0,C 180,E1 -10877.449,E2 -10877.449} C_VEL
LIN {X 0,Y 403.3,Z 862.329,A -85,B 0,C 180,E1 -10879.457,E2 -10879.457} C_VEL
LIN {X 0,Y 403.113,Z 865.938,A -85,B 0,C 180,E1 -10880.973,E2 -10880.973} C_VEL
LIN {X 0,Y 402.974,Z 869.783,A -85,B 0,C 180,E1 -10882.988,E2 -10882.988} C_VEL
LIN {X 0,Y 402.867,Z 872.624,A -85,B 0,C 180,E1 -10884.996,E2 -10884.996} C_VEL
LIN {X 0,Y 402.797,Z 874.499,A -85,B 0,C 180,E1 -10887,E2 -10887} C_VEL
LIN {X 0,Y 402.853,Z 875.174,A -85,B 0,C 180,E1 -10888.001,E2 -10888.001} C_VEL
LIN {X 0,Y 402.81,Z 875.644,A -85,B 0,C 180,E1 -10890,E2 -10890} C_VEL
LIN {X 0,Y 402.853,Z 875.174,A -85,B 0,C 180,E1 -10891.999,E2 -10891.999} C_VEL
LIN {X 0,Y 402.809,Z 873.755,A -85,B 0,C 180,E1 -10894.002,E2 -10894.002} C_VEL
LIN {X 0,Y 402.938,Z 871.102,A -85,B 0,C 180,E1 -10896.182,E2 -10896.182} C_VEL
LIN {X 0,Y 403.062,Z 866.977,A -85,B 0,C 180,E1 -10898.523,E2 -10898.523} C_VEL
LIN {X 0,Y 403.184,Z 863.613,A -85,B 0,C 180,E1 -10900.038,E2 -10900.038} C_VEL
LIN {X 0,Y 403.658,Z 858.121,A -85,B 0,C 180,E1 -10902.059,E2 -10902.059} C_VEL
LIN {X 0,Y 404.123,Z 853.265,A -85,B 0,C 180,E1 -10903.578,E2 -10903.578} C_VEL
LIN {X 0,Y 404.934,Z 845.599,A -85,B 0,C 180,E1 -10905.605,E2 -10905.605} C_VEL
LIN {X 0,Y 405.834,Z 838.95,A -85,B 0,C 180,E1 -10907.121,E2 -10907.121} C_VEL
LIN {X 0,Y 406.717,Z 831.393,A -85,B 0,C 180,E1 -10908.643,E2 -10908.643} C_VEL
LIN {X 0,Y 407.882,Z 822.806,A -85,B 0,C 180,E1 -10910.157,E2 -10910.157} C_VEL
LIN {X 0,Y 409.265,Z 813.325,A -85,B 0,C 180,E1 -10911.62,E2 -10911.62} C_VEL
LIN {X 0,Y 410.72,Z 802.786,A -85,B 0,C 180,E1 -10913.042,E2 -10913.042} C_VEL
LIN {X 0,Y 412.155,Z 792.213,A -85,B 0,C 180,E1 -10914.291,E2 -10914.291} C_VEL
LIN {X 0,Y 413.789,Z 780.892,A -85,B 0,C 180,E1 -10915.447,E2 -10915.447} C_VEL
LIN {X 0,Y 415.125,Z 770.454,A -85,B 0,C 180,E1 -10916.385,E2 -10916.385} C_VEL
LIN {X 0,Y 416.467,Z 759.534,A -85,B 0,C 180,E1 -10917.241,E2 -10917.241} C_VEL
LIN {X 0,Y 417.907,Z 746.798,A -85,B 0,C 180,E1 -10918.091,E2 -10918.091} C_VEL
LIN {X 0,Y 419.182,Z 733.795,A -85,B 0,C 180,E1 -10918.817,E2 -10918.817} C_VEL
LIN {X 0,Y 420.378,Z 720.212,A -85,B 0,C 180,E1 -10919.429,E2 -10919.429} C_VEL
LIN {X 0,Y 421.261,Z 707.163,A -85,B 0,C 180,E1 -10919.896,E2 -10919.896} C_VEL
LIN {X 0,Y 422.012,Z 693.753,A -85,B 0,C 180,E1 -10920.249,E2 -10920.249} C_VEL
LIN {X 0,Y 422.985,Z 656.467,A -85,B 0,C 180,E1 -10920.932,E2 -10920.932} C_VEL
LIN {X 0,Y 426.053,Z 524.514,A -85,B 0,C 180,E1 -10923.25,E2 -10923.25} C_VEL
LIN {X 0,Y 420.202,Z 500.057,A -85,B 0,C 180,E1 -10924.263,E2 -10924.263} C_VEL
LIN {X 0,Y 411.647,Z 482.711,A -85,B 0,C 180,E1 -10925.434,E2 -10925.434} C_VEL
LIN {X 0,Y 410.246,Z 479.566,A -85,B 0,C 180,E1 -10925.679,E2 -10925.679} C_VEL
LIN {X 0,Y 406.997,Z 467.505,A -85,B 0,C 180,E1 -10928.435,E2 -10928.435} C_VEL
LIN {X 0,Y 404.143,Z 457.546,A -85,B 0,C 180,E1 -10930.938,E2 -10930.938} C_VEL
LIN {X 0,Y 404.148,Z 457.395,A -85,B 0,C 180,E1 -10934.073,E2 -10934.073} C_VEL
LIN {X 0,Y 404.201,Z 457.384,A -85,B 0,C 180,E1 -10937.304,E2 -10937.304} C_VEL
LIN {X 0,Y 404.163,Z 457.37,A -85,B 0,C 180,E1 -10939.955,E2 -10939.955} C_VEL
LIN {X 0,Y 404.135,Z 457.393,A -85,B 0,C 180,E1 -10943.124,E2 -10943.124} C_VEL
LIN {X 0,Y 404.139,Z 457.375,A -85,B 0,C 180,E1 -10946.187,E2 -10946.187} C_VEL
LIN {X 0,Y 404.148,Z 457.373,A -85,B 0,C 180,E1 -10949.715,E2 -10949.715} C_VEL
LIN {X 0,Y 404.189,Z 457.36,A -85,B 0,C 180,E1 -10953.122,E2 -10953.122} C_VEL
LIN {X 0,Y 404.167,Z 457.388,A -85,B 0,C 180,E1 -10955.334,E2 -10955.334} C_VEL
LIN {X 0,Y 404.13,Z 457.357,A -85,B 0,C 180,E1 -10958.58,E2 -10958.58} C_VEL
LIN {X 0,Y 404.202,Z 457.358,A -85,B 0,C 180,E1 -10961.761,E2 -10961.761} C_VEL
LIN {X 0,Y 404.198,Z 457.381,A -85,B 0,C 180,E1 -10964.882,E2 -10964.882} C_VEL
LIN {X 0,Y 404.249,Z 457.372,A -85,B 0,C 180,E1 -10967.958,E2 -10967.958} C_VEL
LIN {X 0,Y 404.397,Z 457.348,A -85,B 0,C 180,E1 -10972.128,E2 -10972.128} C_VEL
LIN {X 0,Y 404.426,Z 457.358,A -85,B 0,C 180,E1 -10974.015,E2 -10974.015} C_VEL
LIN {X 0,Y 404.474,Z 457.346,A -85,B 0,C 180,E1 -10978.008,E2 -10978.008} C_VEL
LIN {X 0,Y 404.602,Z 457.333,A -85,B 0,C 180,E1 -10980,E2 -10980} C_VEL
LIN {X 0,Y 404.416,Z 457.356,A -85,B 0,C 180,E1 -10982.988,E2 -10982.988} C_VEL
LIN {X 0,Y 404.388,Z 457.348,A -85,B 0,C 180,E1 -10986.619,E2 -10986.619} C_VEL
LIN {X 0,Y 404.283,Z 457.372,A -85,B 0,C 180,E1 -10989.001,E2 -10989.001} C_VEL
LIN {X 0,Y 404.248,Z 457.368,A -85,B 0,C 180,E1 -10992.041,E2 -10992.041} C_VEL
LIN {X 0,Y 404.197,Z 457.374,A -85,B 0,C 180,E1 -10995.118,E2 -10995.118} C_VEL
LIN {X 0,Y 404.201,Z 457.385,A -85,B 0,C 180,E1 -10998.238,E2 -10998.238} C_VEL
LIN {X 0,Y 404.129,Z 457.392,A -85,B 0,C 180,E1 -11001.419,E2 -11001.419} C_VEL
LIN {X 0,Y 404.166,Z 457.369,A -85,B 0,C 180,E1 -11004.666,E2 -11004.666} C_VEL
LIN {X 0,Y 404.19,Z 457.356,A -85,B 0,C 180,E1 -11008,E2 -11008} C_VEL
LIN {X 0,Y 404.135,Z 457.388,A -85,B 0,C 180,E1 -11011.559,E2 -11011.559} C_VEL
LIN {X 0,Y 404.177,Z 457.355,A -85,B 0,C 180,E1 -11015.016,E2 -11015.016} C_VEL
LIN {X 0,Y 404.157,Z 457.393,A -85,B 0,C 180,E1 -11018.756,E2 -11018.756} C_VEL
LIN {X 0,Y 404.184,Z 457.39,A -85,B 0,C 180,E1 -11021.611,E2 -11021.611} C_VEL
LIN {X 0,Y 404.186,Z 457.388,A -85,B 0,C 180,E1 -11024.529,E2 -11024.529} C_VEL
LIN {X 0,Y 404.164,Z 457.392,A -85,B 0,C 180,E1 -11027.3,E2 -11027.3} C_VEL
LIN {X 0,Y 404.162,Z 457.39,A -85,B 0,C 180,E1 -11029.956,E2 -11029.956} C_VEL
LIN {X 0,Y 404.134,Z 457.395,A -85,B 0,C 180,E1 -11033.125,E2 -11033.125} C_VEL
LIN {X 0,Y 404.139,Z 457.395,A -85,B 0,C 180,E1 -11036.188,E2 -11036.188} C_VEL
LIN {X 0,Y 404.14,Z 457.394,A -85,B 0,C 180,E1 -11039.715,E2 -11039.715} C_VEL
LIN {X 0,Y 404.19,Z 457.387,A -85,B 0,C 180,E1 -11043.123,E2 -11043.123} C_VEL
LIN {X 0,Y 404.173,Z 457.391,A -85,B 0,C 180,E1 -11045.335,E2 -11045.335} C_VEL
LIN {X 0,Y 404.134,Z 457.393,A -85,B 0,C 180,E1 -11048.581,E2 -11048.581} C_VEL
LIN {X 0,Y 404.206,Z 457.387,A -85,B 0,C 180,E1 -11051.762,E2 -11051.762} C_VEL
LIN {X 0,Y 404.204,Z 457.388,A -85,B 0,C 180,E1 -11054.882,E2 -11054.882} C_VEL
LIN {X 0,Y 404.266,Z 457.378,A -85,B 0,C 180,E1 -11057.959,E2 -11057.959} C_VEL
LIN {X 0,Y 404.43,Z 457.358,A -85,B 0,C 180,E1 -11062.1,E2 -11062.1} C_VEL
LIN {X 0,Y 404.42,Z 457.359,A -85,B 0,C 180,E1 -11064.015,E2 -11064.015} C_VEL
LIN {X 0,Y 404.48,Z 457.351,A -85,B 0,C 180,E1 -11068.009,E2 -11068.009} C_VEL
LIN {X 0,Y 404.608,Z 457.339,A -85,B 0,C 180,E1 -11070,E2 -11070} C_VEL
LIN {X 0,Y 404.42,Z 457.36,A -85,B 0,C 180,E1 -11072.988,E2 -11072.988} C_VEL
LIN {X 0,Y 404.408,Z 457.362,A -85,B 0,C 180,E1 -11076.987,E2 -11076.987} C_VEL
LIN {X 0,Y 404.267,Z 457.378,A -85,B 0,C 180,E1 -11080.011,E2 -11080.011} C_VEL
LIN {X 0,Y 404.263,Z 457.378,A -85,B 0,C 180,E1 -11083.211,E2 -11083.211} C_VEL
LIN {X 0,Y 404.212,Z 457.384,A -85,B 0,C 180,E1 -11087.007,E2 -11087.007} C_VEL
LIN {X 0,Y 404.159,Z 457.392,A -85,B 0,C 180,E1 -11090.351,E2 -11090.351} C_VEL
LIN {X 0,Y 404.131,Z 457.392,A -85,B 0,C 180,E1 -11091.927,E2 -11091.927} C_VEL
LIN {X 0,Y 403.49,Z 457.476,A -85,B 0,C 180,E1 -11092.758,E2 -11092.758} C_VEL
LIN {X 0,Y 400.657,Z 457.834,A -85,B 0,C 180,E1 -11094.11,E2 -11094.11} C_VEL
LIN {X 0,Y 398.247,Z 458.135,A -85,B 0,C 180,E1 -11095.202,E2 -11095.202} C_VEL
LIN {X 0,Y 397.213,Z 458.26,A -85,B 0,C 180,E1 -11096.047,E2 -11096.047} C_VEL
LIN {X 0,Y 397.129,Z 458.268,A -85,B 0,C 180,E1 -11096.332,E2 -11096.332} C_VEL
LIN {X 0,Y 397.117,Z 458.269,A -85,B 0,C 180,E1 -11098.543,E2 -11098.543} C_VEL
LIN {X 0,Y 397.073,Z 458.276,A -85,B 0,C 180,E1 -11102.071,E2 -11102.071} C_VEL
LIN {X 0,Y 397.114,Z 458.267,A -85,B 0,C 180,E1 -11105.503,E2 -11105.503} C_VEL
LIN {X 0,Y 397.131,Z 458.268,A -85,B 0,C 180,E1 -11108.862,E2 -11108.862} C_VEL
LIN {X 0,Y 397.107,Z 458.271,A -85,B 0,C 180,E1 -11112.261,E2 -11112.261} C_VEL
LIN {X 0,Y 397.158,Z 458.266,A -85,B 0,C 180,E1 -11116.36,E2 -11116.36} C_VEL
LIN {X 0,Y 397.117,Z 458.269,A -85,B 0,C 180,E1 -11119.55,E2 -11119.55} C_VEL
LIN {X 0,Y 397.116,Z 458.272,A -85,B 0,C 180,E1 -11122.785,E2 -11122.785} C_VEL
LIN {X 0,Y 397.11,Z 458.228,A -85,B 0,C 180,E1 -11126.282,E2 -11126.282} C_VEL
LIN {X 0,Y 397.106,Z 458.268,A -85,B 0,C 180,E1 -11130.133,E2 -11130.133} C_VEL
LIN {X 0,Y 397.186,Z 458.217,A -85,B 0,C 180,E1 -11132.61,E2 -11132.61} C_VEL
LIN {X 0,Y 397.12,Z 458.261,A -85,B 0,C 180,E1 -11135.981,E2 -11135.981} C_VEL
LIN {X 0,Y 397.13,Z 458.255,A -85,B 0,C 180,E1 -11139.705,E2 -11139.705} C_VEL
LIN {X 0,Y 397.173,Z 458.258,A -85,B 0,C 180,E1 -11142.845,E2 -11142.845} C_VEL
LIN {X 0,Y 397.22,Z 458.253,A -85,B 0,C 180,E1 -11146.703,E2 -11146.703} C_VEL
LIN {X 0,Y 397.21,Z 458.249,A -85,B 0,C 180,E1 -11149.809,E2 -11149.809} C_VEL
LIN {X 0,Y 397.345,Z 458.229,A -85,B 0,C 180,E1 -11152.888,E2 -11152.888} C_VEL
LIN {X 0,Y 397.25,Z 458.243,A -85,B 0,C 180,E1 -11154.925,E2 -11154.925} C_VEL
LIN {X 0,Y 397.443,Z 458.212,A -85,B 0,C 180,E1 -11157.973,E2 -11157.973} C_VEL
LIN {X 0,Y 397.572,Z 458.209,A -85,B 0,C 180,E1 -11160,E2 -11160} C_VEL
LIN {X 0,Y 397.374,Z 458.226,A -85,B 0,C 180,E1 -11163.042,E2 -11163.042} C_VEL
LIN {X 0,Y 397.375,Z 458.235,A -85,B 0,C 180,E1 -11166.092,E2 -11166.092} C_VEL
LIN {X 0,Y 397.245,Z 458.236,A -85,B 0,C 180,E1 -11169.162,E2 -11169.162} C_VEL
LIN {X 0,Y 397.212,Z 458.246,A -85,B 0,C 180,E1 -11172.258,E2 -11172.258} C_VEL
LIN {X 0,Y 397.171,Z 458.259,A -85,B 0,C 180,E1 -11175.392,E2 -11175.392} C_VEL
LIN {X 0,Y 397.154,Z 458.228,A -85,B 0,C 180,E1 -11178.574,E2 -11178.574} C_VEL
LIN {X 0,Y 397.088,Z 458.24,A -85,B 0,C 180,E1 -11181.819,E2 -11181.819} C_VEL
LIN {X 0,Y 397.146,Z 458.259,A -85,B 0,C 180,E1 -11185.513,E2 -11185.513} C_VEL
LIN {X 0,Y 397.119,Z 458.224,A -85,B 0,C 180,E1 -11188.544,E2 -11188.544} C_VEL
LIN {X 0,Y 397.105,Z 458.273,A -85,B 0,C 180,E1 -11192.069,E2 -11192.069} C_VEL
LIN {X 0,Y 397.114,Z 458.242,A -85,B 0,C 180,E1 -11195.504,E2 -11195.504} C_VEL
LIN {X 0,Y 397.132,Z 458.256,A -85,B 0,C 180,E1 -11198.863,E2 -11198.863} C_VEL
LIN {X 0,Y 397.153,Z 458.267,A -85,B 0,C 180,E1 -11202.256,E2 -11202.256} C_VEL
LIN {X 0,Y 397.106,Z 458.258,A -85,B 0,C 180,E1 -11205.066,E2 -11205.066} C_VEL
LIN {X 0,Y 397.097,Z 458.339,A -85,B 0,C 180,E1 -11208.376,E2 -11208.376} C_VEL
LIN {X 0,Y 397.581,Z 460.156,A -85,B 0,C 180,E1 -11208.93,E2 -11208.93} C_VEL
LIN {X 0,Y 400.751,Z 471.204,A -85,B 0,C 180,E1 -11211.7,E2 -11211.7} C_VEL
LIN {X 0,Y 402.939,Z 479.354,A -85,B 0,C 180,E1 -11213.583,E2 -11213.583} C_VEL
LIN {X 0,Y 411.558,Z 496.596,A -85,B 0,C 180,E1 -11214.847,E2 -11214.847} C_VEL
LIN {X 0,Y 414.846,Z 503.793,A -85,B 0,C 180,E1 -11215.312,E2 -11215.312} C_VEL
LIN {X 0,Y 420.115,Z 526.053,A -85,B 0,C 180,E1 -11216.253,E2 -11216.253} C_VEL
LIN {X 0,Y 416.319,Z 679.541,A -85,B 0,C 180,E1 -11218.976,E2 -11218.976} C_VEL
LIN {X 0,Y 415.507,Z 701,A -85,B 0,C 180,E1 -11219.438,E2 -11219.438} C_VEL
LIN {X 0,Y 414.458,Z 715.753,A -85,B 0,C 180,E1 -11219.914,E2 -11219.914} C_VEL
LIN {X 0,Y 413.424,Z 728.646,A -85,B 0,C 180,E1 -11220.464,E2 -11220.464} C_VEL
LIN {X 0,Y 412.166,Z 741.455,A -85,B 0,C 180,E1 -11221.134,E2 -11221.134} C_VEL
LIN {X 0,Y 410.775,Z 754.097,A -85,B 0,C 180,E1 -11221.934,E2 -11221.934} C_VEL
LIN {X 0,Y 409.319,Z 765.741,A -85,B 0,C 180,E1 -11222.797,E2 -11222.797} C_VEL
LIN {X 0,Y 407.81,Z 777.269,A -85,B 0,C 180,E1 -11223.794,E2 -11223.794} C_VEL
LIN {X 0,Y 406.156,Z 788.569,A -85,B 0,C 180,E1 -11224.917,E2 -11224.917} C_VEL
LIN {X 0,Y 404.553,Z 799.552,A -85,B 0,C 180,E1 -11226.178,E2 -11226.178} C_VEL
LIN {X 0,Y 403.015,Z 809.993,A -85,B 0,C 180,E1 -11227.554,E2 -11227.554} C_VEL
LIN {X 0,Y 401.573,Z 819.459,A -85,B 0,C 180,E1 -11228.976,E2 -11228.976} C_VEL
LIN {X 0,Y 400.235,Z 828.42,A -85,B 0,C 180,E1 -11230.511,E2 -11230.511} C_VEL
LIN {X 0,Y 399.142,Z 836.473,A -85,B 0,C 180,E1 -11232.088,E2 -11232.088} C_VEL
LIN {X 0,Y 398.299,Z 843.281,A -85,B 0,C 180,E1 -11233.602,E2 -11233.602} C_VEL
LIN {X 0,Y 397.541,Z 849.421,A -85,B 0,C 180,E1 -11235.147,E2 -11235.147} C_VEL
LIN {X 0,Y 396.801,Z 856.633,A -85,B 0,C 180,E1 -11237.299,E2 -11237.299} C_VEL
LIN {X 0,Y 396.255,Z 862.117,A -85,B 0,C 180,E1 -11239.268,E2 -11239.268} C_VEL
LIN {X 0,Y 396.024,Z 865.726,A -85,B 0,C 180,E1 -11240.81,E2 -11240.81} C_VEL
LIN {X 0,Y 395.894,Z 869.572,A -85,B 0,C 180,E1 -11242.862,E2 -11242.862} C_VEL
LIN {X 0,Y 395.768,Z 872.414,A -85,B 0,C 180,E1 -11244.906,E2 -11244.906} C_VEL
LIN {X 0,Y 395.732,Z 873.545,A -85,B 0,C 180,E1 -11245.926,E2 -11245.926} C_VEL
LIN {X 0,Y 395.751,Z 874.964,A -85,B 0,C 180,E1 -11247.965,E2 -11247.965} C_VEL
LIN {X 0,Y 395.74,Z 875.435,A -85,B 0,C 180,E1 -11250,E2 -11250} C_VEL
LIN {X 0,Y 395.751,Z 874.964,A -85,B 0,C 180,E1 -11252.035,E2 -11252.035} C_VEL
LIN {X 0,Y 395.732,Z 873.545,A -85,B 0,C 180,E1 -11254.074,E2 -11254.074} C_VEL
LIN {X 0,Y 395.857,Z 871.089,A -85,B 0,C 180,E1 -11256.166,E2 -11256.166} C_VEL
LIN {X 0,Y 395.988,Z 866.765,A -85,B 0,C 180,E1 -11258.676,E2 -11258.676} C_VEL
LIN {X 0,Y 396.121,Z 863.401,A -85,B 0,C 180,E1 -11260.219,E2 -11260.219} C_VEL
LIN {X 0,Y 396.639,Z 857.909,A -85,B 0,C 180,E1 -11262.276,E2 -11262.276} C_VEL
LIN {X 0,Y 397.126,Z 853.053,A -85,B 0,C 180,E1 -11263.822,E2 -11263.822} C_VEL
LIN {X 0,Y 397.998,Z 845.386,A -85,B 0,C 180,E1 -11265.884,E2 -11265.884} C_VEL
LIN {X 0,Y 398.899,Z 838.736,A -85,B 0,C 180,E1 -11267.428,E2 -11267.428} C_VEL
LIN {X 0,Y 399.862,Z 831.179,A -85,B 0,C 180,E1 -11268.975,E2 -11268.975} C_VEL
LIN {X 0,Y 401.083,Z 822.592,A -85,B 0,C 180,E1 -11270.514,E2 -11270.514} C_VEL
LIN {X 0,Y 402.505,Z 813.504,A -85,B 0,C 180,E1 -11271.942,E2 -11271.942} C_VEL
LIN {X 0,Y 404.063,Z 802.572,A -85,B 0,C 180,E1 -11273.445,E2 -11273.445} C_VEL
LIN {X 0,Y 405.607,Z 792,A -85,B 0,C 180,E1 -11274.709,E2 -11274.709} C_VEL
LIN {X 0,Y 407.148,Z 781.926,A -85,B 0,C 180,E1 -11275.761,E2 -11275.761} C_VEL
LIN {X 0,Y 408.725,Z 770.243,A -85,B 0,C 180,E1 -11276.831,E2 -11276.831} C_VEL
LIN {X 0,Y 410.303,Z 757.579,A -85,B 0,C 180,E1 -11277.823,E2 -11277.823} C_VEL
LIN {X 0,Y 411.777,Z 745.562,A -85,B 0,C 180,E1 -11278.617,E2 -11278.617} C_VEL
LIN {X 0,Y 412.95,Z 733.585,A -85,B 0,C 180,E1 -11279.294,E2 -11279.294} C_VEL
LIN {X 0,Y 414.155,Z 720.251,A -85,B 0,C 180,E1 -11279.904,E2 -11279.904} C_VEL
LIN {X 0,Y 415.081,Z 707.401,A -85,B 0,C 180,E1 -11280.372,E2 -11280.372} C_VEL
LIN {X 0,Y 415.891,Z 693.543,A -85,B 0,C 180,E1 -11280.742,E2 -11280.742} C_VEL
LIN {X 0,Y 416.907,Z 656.257,A -85,B 0,C 180,E1 -11281.434,E2 -11281.434} C_VEL
LIN {X 0,Y 420.105,Z 526.077,A -85,B 0,C 180,E1 -11283.748,E2 -11283.748} C_VEL
LIN {X 0,Y 414.748,Z 503.362,A -85,B 0,C 180,E1 -11284.706,E2 -11284.706} C_VEL
LIN {X 0,Y 406.827,Z 487.123,A -85,B 0,C 180,E1 -11285.821,E2 -11285.821} C_VEL
LIN {X 0,Y 403.058,Z 479.491,A -85,B 0,C 180,E1 -11286.393,E2 -11286.393} C_VEL
LIN {X 0,Y 400.021,Z 468.431,A -85,B 0,C 180,E1 -11288.975,E2 -11288.975} C_VEL
LIN {X 0,Y 397.115,Z 458.51,A -85,B 0,C 180,E1 -11291.527,E2 -11291.527} C_VEL
LIN {X 0,Y 397.063,Z 458.262,A -85,B 0,C 180,E1 -11292.267,E2 -11292.267} C_VEL
LIN {X 0,Y 397.111,Z 458.256,A -85,B 0,C 180,E1 -11295.064,E2 -11295.064} C_VEL
LIN {X 0,Y 397.15,Z 458.265,A -85,B 0,C 180,E1 -11298.006,E2 -11298.006} C_VEL
LIN {X 0,Y 397.104,Z 458.266,A -85,B 0,C 180,E1 -11301.725,E2 -11301.725} C_VEL
LIN {X 0,Y 397.119,Z 458.24,A -85,B 0,C 180,E1 -11305.506,E2 -11305.506} C_VEL
LIN {X 0,Y 397.081,Z 458.267,A -85,B 0,C 180,E1 -11309.118,E2 -11309.118} C_VEL
LIN {X 0,Y 397.188,Z 458.221,A -85,B 0,C 180,E1 -11312.609,E2 -11312.609} C_VEL
LIN {X 0,Y 397.122,Z 458.269,A -85,B 0,C 180,E1 -11315.981,E2 -11315.981} C_VEL
LIN {X 0,Y 397.131,Z 458.214,A -85,B 0,C 180,E1 -11319.704,E2 -11319.704} C_VEL
LIN {X 0,Y 397.174,Z 458.251,A -85,B 0,C 180,E1 -11322.844,E2 -11322.844} C_VEL
LIN {X 0,Y 397.221,Z 458.241,A -85,B 0,C 180,E1 -11326.702,E2 -11326.702} C_VEL
LIN {X 0,Y 397.21,Z 458.255,A -85,B 0,C 180,E1 -11329.809,E2 -11329.809} C_VEL
LIN {X 0,Y 397.344,Z 458.239,A -85,B 0,C 180,E1 -11332.888,E2 -11332.888} C_VEL
LIN {X 0,Y 397.251,Z 458.246,A -85,B 0,C 180,E1 -11334.925,E2 -11334.925} C_VEL
LIN {X 0,Y 397.443,Z 458.222,A -85,B 0,C 180,E1 -11337.973,E2 -11337.973} C_VEL
LIN {X 0,Y 397.572,Z 458.208,A -85,B 0,C 180,E1 -11340,E2 -11340} C_VEL
LIN {X 0,Y 397.374,Z 458.233,A -85,B 0,C 180,E1 -11343.041,E2 -11343.041} C_VEL
LIN {X 0,Y 397.34,Z 458.225,A -85,B 0,C 180,E1 -11346.616,E2 -11346.616} C_VEL
LIN {X 0,Y 397.244,Z 458.247,A -85,B 0,C 180,E1 -11349.162,E2 -11349.162} C_VEL
LIN {X 0,Y 397.211,Z 458.246,A -85,B 0,C 180,E1 -11352.258,E2 -11352.258} C_VEL
LIN {X 0,Y 397.17,Z 458.246,A -85,B 0,C 180,E1 -11355.392,E2 -11355.392} C_VEL
LIN {X 0,Y 397.154,Z 458.266,A -85,B 0,C 180,E1 -11358.573,E2 -11358.573} C_VEL
LIN {X 0,Y 397.087,Z 458.269,A -85,B 0,C 180,E1 -11361.819,E2 -11361.819} C_VEL
LIN {X 0,Y 397.144,Z 458.228,A -85,B 0,C 180,E1 -11365.512,E2 -11365.512} C_VEL
LIN {X 0,Y 397.119,Z 458.248,A -85,B 0,C 180,E1 -11368.543,E2 -11368.543} C_VEL
LIN {X 0,Y 397.073,Z 458.261,A -85,B 0,C 180,E1 -11372.072,E2 -11372.072} C_VEL
LIN {X 0,Y 397.112,Z 458.243,A -85,B 0,C 180,E1 -11375.504,E2 -11375.504} C_VEL
LIN {X 0,Y 397.13,Z 458.269,A -85,B 0,C 180,E1 -11378.863,E2 -11378.863} C_VEL
LIN {X 0,Y 397.153,Z 458.264,A -85,B 0,C 180,E1 -11382.255,E2 -11382.255} C_VEL
LIN {X 0,Y 397.105,Z 458.272,A -85,B 0,C 180,E1 -11385.065,E2 -11385.065} C_VEL
LIN {X 0,Y 397.103,Z 458.27,A -85,B 0,C 180,E1 -11388.015,E2 -11388.015} C_VEL
LIN {X 0,Y 397.131,Z 458.268,A -85,B 0,C 180,E1 -11391.138,E2 -11391.138} C_VEL
LIN {X 0,Y 397.114,Z 458.267,A -85,B 0,C 180,E1 -11394.497,E2 -11394.497} C_VEL
LIN {X 0,Y 397.073,Z 458.276,A -85,B 0,C 180,E1 -11397.929,E2 -11397.929} C_VEL
LIN {X 0,Y 397.117,Z 458.268,A -85,B 0,C 180,E1 -11401.457,E2 -11401.457} C_VEL
LIN {X 0,Y 397.148,Z 458.263,A -85,B 0,C 180,E1 -11404.488,E2 -11404.488} C_VEL
LIN {X 0,Y 397.105,Z 458.269,A -85,B 0,C 180,E1 -11407.086,E2 -11407.086} C_VEL
